LIN {X 0.147,Y -413.932,Z 942.824,A 0.000,B 0.000,C 90.000,E1 4.302} C_DIS
LIN {X -0.071,Y -420.578,Z 942.807,A 0.000,B 0.000,C 90.000,E1 1.260} C_DIS
LIN {X -0.166,Y -425.869,Z 942.795,A 0.000,B 0.000,C 90.000,E1 359.141} C_DIS
LIN {X 0.033,Y -428.792,Z 942.791,A 0.000,B 0.000,C 90.000,E1 358.282} C_DIS
LIN {X 0.078,Y -429.567,Z 942.790,A 0.000,B 0.000,C 90.000,E1 358.108} C_DIS
LIN {X -0.181,Y -431.033,Z 942.788,A 0.000,B 0.000,C 90.000,E1 357.879} C_DIS
LIN {X -0.110,Y -433.741,Z 942.786,A 0.000,B 0.000,C 90.000,E1 357.535} C_DIS
LIN {X -0.183,Y -435.827,Z 942.785,A 0.000,B 0.000,C 90.000,E1 357.306} C_DIS
LIN {X -0.171,Y -439.740,Z 942.783,A 0.000,B 0.000,C 90.000,E1 357.020} C_DIS
LIN {X -0.164,Y -441.464,Z 942.783,A 0.000,B 0.000,C 90.000,E1 356.906} C_DIS
LIN {X 0.019,Y -456.050,Z 942.779,A 0.000,B 0.000,C 90.000,E1 356.159} C_DIS
LIN {X -0.206,Y -464.593,Z 942.776,A 0.000,B 0.000,C 90.000,E1 355.755} C_DIS
LIN {X 0.207,Y -481.185,Z 942.771,A 0.000,B 0.000,C 90.000,E1 354.837} C_DIS
LIN {X 0.033,Y -494.438,Z 942.768,A 0.000,B 0.000,C 90.000,E1 354.147} C_DIS
LIN {X 0.171,Y -504.283,Z 942.764,A 0.000,B 0.000,C 90.000,E1 353.571} C_DIS
LIN {X -0.140,Y -515.374,Z 942.761,A 0.000,B 0.000,C 90.000,E1 352.932} C_DIS
LIN {X -0.046,Y -523.150,Z 942.758,A 0.000,B 0.000,C 90.000,E1 352.413} C_DIS
LIN {X -0.040,Y -531.958,Z 942.754,A 0.000,B 0.000,C 90.000,E1 351.781} C_DIS
LIN {X 0.025,Y -539.240,Z 942.751,A 0.000,B 0.000,C 90.000,E1 351.197} C_DIS
LIN {X -0.295,Y -546.239,Z 942.748,A 0.000,B 0.000,C 90.000,E1 350.622} C_DIS
LIN {X -0.106,Y -551.498,Z 942.745,A 0.000,B 0.000,C 90.000,E1 350.095} C_DIS
LIN {X 0.210,Y -557.779,Z 942.741,A 0.000,B 0.000,C 90.000,E1 349.398} C_DIS
LIN {X -0.265,Y -563.672,Z 942.737,A 0.000,B 0.000,C 90.000,E1 348.757} C_DIS
LIN {X 0.059,Y -568.140,Z 942.734,A 0.000,B 0.000,C 90.000,E1 348.173} C_DIS
LIN {X -0.068,Y -575.153,Z 942.729,A 0.000,B 0.000,C 90.000,E1 347.229} C_DIS
LIN {X 0.103,Y -579.773,Z 942.725,A 0.000,B 0.000,C 90.000,E1 346.533} C_DIS
LIN {X 0.025,Y -586.493,Z 942.719,A 0.000,B 0.000,C 90.000,E1 345.463} C_DIS
LIN {X 0.044,Y -592.545,Z 942.713,A 0.000,B 0.000,C 90.000,E1 344.393} C_DIS
LIN {X 0.209,Y -597.463,Z 942.708,A 0.000,B 0.000,C 90.000,E1 343.449} C_DIS
LIN {X 0.026,Y -601.982,Z 942.703,A 0.000,B 0.000,C 90.000,E1 342.543} C_DIS
LIN {X -0.139,Y -606.953,Z 942.697,A 0.000,B 0.000,C 90.000,E1 341.511} C_DIS
LIN {X -0.175,Y -610.557,Z 942.693,A 0.000,B 0.000,C 90.000,E1 340.732} C_DIS
LIN {X 0.025,Y -613.980,Z 942.689,A 0.000,B 0.000,C 90.000,E1 339.934} C_DIS
LIN {X 0.013,Y -618.273,Z 942.683,A 0.000,B 0.000,C 90.000,E1 338.901} C_DIS
LIN {X 0.283,Y -622.282,Z 942.677,A 0.000,B 0.000,C 90.000,E1 337.847} C_DIS
LIN {X 0.035,Y -626.049,Z 942.671,A 0.000,B 0.000,C 90.000,E1 336.847} C_DIS
LIN {X -0.400,Y -630.401,Z 942.664,A 0.000,B 0.000,C 90.000,E1 335.613} C_DIS
LIN {X 0.327,Y -634.450,Z 942.657,A 0.000,B 0.000,C 90.000,E1 334.280} C_DIS
LIN {X -0.012,Y -638.192,Z 942.650,A 0.000,B 0.000,C 90.000,E1 333.050} C_DIS
LIN {X 0.220,Y -640.863,Z 942.645,A 0.000,B 0.000,C 90.000,E1 332.025} C_DIS
LIN {X -0.152,Y -642.800,Z 942.641,A 0.000,B 0.000,C 90.000,E1 331.307} C_DIS
LIN {X 0.034,Y -646.291,Z 942.632,A 0.000,B 0.000,C 90.000,E1 329.793} C_DIS
LIN {X 0.199,Y -648.852,Z 942.625,A 0.000,B 0.000,C 90.000,E1 328.535} C_DIS
LIN {X 0.231,Y -650.232,Z 942.621,A 0.000,B 0.000,C 90.000,E1 327.788} C_DIS
LIN {X -0.186,Y -651.837,Z 942.616,A 0.000,B 0.000,C 90.000,E1 326.834} C_DIS
LIN {X -0.140,Y -653.569,Z 942.609,A 0.000,B 0.000,C 90.000,E1 325.595} C_DIS
LIN {X -0.149,Y -654.821,Z 942.603,A 0.000,B 0.000,C 90.000,E1 324.609} C_DIS
LIN {X -0.141,Y -655.872,Z 942.598,A 0.000,B 0.000,C 90.000,E1 323.623} C_DIS
LIN {X 0.286,Y -657.151,Z 942.590,A 0.000,B 0.000,C 90.000,E1 322.110} C_DIS
LIN {X -0.238,Y -658.485,Z 942.580,A 0.000,B 0.000,C 90.000,E1 320.436} C_DIS
LIN {X 0.159,Y -659.046,Z 942.576,A 0.000,B 0.000,C 90.000,E1 319.666} C_DIS
LIN {X 0.057,Y -660.436,Z 942.565,A 0.000,B 0.000,C 90.000,E1 317.715} C_DIS
LIN {X -0.058,Y -661.637,Z 942.557,A 0.000,B 0.000,C 90.000,E1 316.257} C_DIS
LIN {X 0.373,Y -662.239,Z 942.553,A 0.000,B 0.000,C 90.000,E1 315.486} C_DIS
LIN {X -0.195,Y -664.346,Z 942.539,A 0.000,B 0.000,C 90.000,E1 313.095} C_DIS
LIN {X -0.202,Y -665.986,Z 942.530,A 0.000,B 0.000,C 90.000,E1 311.391} C_DIS
LIN {X -0.170,Y -667.075,Z 942.523,A 0.000,B 0.000,C 90.000,E1 310.172} C_DIS
LIN {X -0.041,Y -668.319,Z 942.515,A 0.000,B 0.000,C 90.000,E1 308.705} C_DIS
LIN {X -0.404,Y -669.174,Z 942.508,A 0.000,B 0.000,C 90.000,E1 307.523} C_DIS
LIN {X 0.209,Y -669.600,Z 942.504,A 0.000,B 0.000,C 90.000,E1 306.744} C_DIS
LIN {X 0.390,Y -670.030,Z 942.498,A 0.000,B 0.000,C 90.000,E1 305.518} C_DIS
LIN {X 0.009,Y -670.808,Z 942.485,A 0.000,B 0.000,C 90.000,E1 303.372} C_DIS
LIN {X -0.049,Y -671.525,Z 942.477,A 0.000,B 0.000,C 90.000,E1 301.926} C_DIS
LIN {X -0.135,Y -675.368,Z 942.453,A 0.000,B 0.000,C 90.000,E1 297.590} C_DIS
LIN {X -0.137,Y -678.486,Z 942.443,A 0.000,B 0.000,C 90.000,E1 295.668} C_DIS
LIN {X -0.057,Y -680.495,Z 942.436,A 0.000,B 0.000,C 90.000,E1 294.463} C_DIS
LIN {X 0.046,Y -682.176,Z 942.429,A 0.000,B 0.000,C 90.000,E1 293.259} C_DIS
LIN {X 0.384,Y -682.822,Z 942.425,A 0.000,B 0.000,C 90.000,E1 292.514} C_DIS
LIN {X -0.104,Y -682.320,Z 942.423,A 0.000,B 0.000,C 90.000,E1 292.078} C_DIS
LIN {X -0.159,Y -681.925,Z 942.421,A 0.000,B 0.000,C 90.000,E1 291.844} C_DIS
LIN {X 0.038,Y -680.853,Z 942.420,A 0.000,B 0.000,C 90.000,E1 291.589} C_DIS
LIN {X 0.079,Y -678.846,Z 942.418,A 0.000,B 0.000,C 90.000,E1 291.227} C_DIS
LIN {X 0.172,Y -678.042,Z 942.417,A 0.000,B 0.000,C 90.000,E1 291.099} C_DIS
LIN {X 0.263,Y -676.847,Z 942.417,A 0.000,B 0.000,C 90.000,E1 290.972} C_DIS
LIN {X -0.270,Y -673.855,Z 942.415,A 0.000,B 0.000,C 90.000,E1 290.791} C_DIS
LIN {X -0.145,Y -669.235,Z 942.414,A 0.000,B 0.000,C 90.000,E1 290.482} C_DIS
LIN {X -0.196,Y -666.122,Z 942.413,A 0.000,B 0.000,C 90.000,E1 290.301} C_DIS
LIN {X 0.016,Y -663.674,Z 942.412,A 0.000,B 0.000,C 90.000,E1 290.120} C_DIS
LIN {X 0.198,Y -661.585,Z 942.411,A 0.000,B 0.000,C 90.000,E1 289.939} C_DIS
LIN {X 0.134,Y -661.564,Z 942.411,A 0.000,B 0.000,C 90.000,E1 289.939} C_DIS
LIN {X 0.203,Y -661.139,Z 942.410,A 0.000,B 0.000,C 90.000,E1 289.812} C_DIS
LIN {X 0.209,Y -661.461,Z 942.409,A 0.000,B 0.000,C 90.000,E1 289.523} C_DIS
LIN {X 0.322,Y -662.225,Z 942.407,A 0.000,B 0.000,C 90.000,E1 289.268} C_DIS
LIN {X 0.275,Y -663.656,Z 942.405,A 0.000,B 0.000,C 90.000,E1 288.906} C_DIS
LIN {X 0.104,Y -670.753,Z 942.398,A 0.000,B 0.000,C 90.000,E1 287.583} C_DIS
LIN {X 0.162,Y -673.111,Z 942.395,A 0.000,B 0.000,C 90.000,E1 287.094} C_DIS
LIN {X -0.022,Y -676.230,Z 942.391,A 0.000,B 0.000,C 90.000,E1 286.386} C_DIS
LIN {X 0.015,Y -678.639,Z 942.387,A 0.000,B 0.000,C 90.000,E1 285.662} C_DIS
LIN {X -0.071,Y -680.054,Z 942.384,A 0.000,B 0.000,C 90.000,E1 285.190} C_DIS
LIN {X -0.181,Y -681.680,Z 942.380,A 0.000,B 0.000,C 90.000,E1 284.481} C_DIS
LIN {X -0.301,Y -683.543,Z 942.375,A 0.000,B 0.000,C 90.000,E1 283.536} C_DIS
LIN {X 0.289,Y -684.620,Z 942.371,A 0.000,B 0.000,C 90.000,E1 282.771} C_DIS
LIN {X 0.197,Y -685.705,Z 942.366,A 0.000,B 0.000,C 90.000,E1 281.827} C_DIS
LIN {X -0.004,Y -685.932,Z 942.362,A 0.000,B 0.000,C 90.000,E1 281.130} C_DIS
LIN {X -0.048,Y -685.875,Z 942.359,A 0.000,B 0.000,C 90.000,E1 280.658} C_DIS
LIN {X -0.219,Y -685.455,Z 942.357,A 0.000,B 0.000,C 90.000,E1 280.197} C_DIS
LIN {X -0.271,Y -684.611,Z 942.354,A 0.000,B 0.000,C 90.000,E1 279.726} C_DIS
LIN {X 0.260,Y -684.093,Z 942.353,A 0.000,B 0.000,C 90.000,E1 279.443} C_DIS
LIN {X 0.195,Y -682.770,Z 942.350,A 0.000,B 0.000,C 90.000,E1 278.973} C_DIS
LIN {X 0.013,Y -681.051,Z 942.347,A 0.000,B 0.000,C 90.000,E1 278.511} C_DIS
LIN {X -0.177,Y -678.961,Z 942.345,A 0.000,B 0.000,C 90.000,E1 278.049} C_DIS
LIN {X 0.087,Y -673.637,Z 942.339,A 0.000,B 0.000,C 90.000,E1 276.947} C_DIS
LIN {X -0.232,Y -670.321,Z 942.335,A 0.000,B 0.000,C 90.000,E1 276.372} C_DIS
LIN {X 0.089,Y -666.532,Z 942.332,A 0.000,B 0.000,C 90.000,E1 275.739} C_DIS
LIN {X -0.194,Y -663.162,Z 942.329,A 0.000,B 0.000,C 90.000,E1 275.277} C_DIS
LIN {X 0.159,Y -659.351,Z 942.327,A 0.000,B 0.000,C 90.000,E1 274.759} C_DIS
LIN {X -0.319,Y -653.995,Z 942.323,A 0.000,B 0.000,C 90.000,E1 274.188} C_DIS
LIN {X -0.137,Y -648.110,Z 942.320,A 0.000,B 0.000,C 90.000,E1 273.555} C_DIS
LIN {X 0.241,Y -644.469,Z 942.318,A 0.000,B 0.000,C 90.000,E1 273.154} C_DIS
LIN {X 0.040,Y -637.861,Z 942.314,A 0.000,B 0.000,C 90.000,E1 272.579} C_DIS
LIN {X 0.156,Y -631.004,Z 942.311,A 0.000,B 0.000,C 90.000,E1 272.007} C_DIS
LIN {X 0.012,Y -623.443,Z 942.308,A 0.000,B 0.000,C 90.000,E1 271.489} C_DIS
LIN {X 0.226,Y -615.726,Z 942.306,A 0.000,B 0.000,C 90.000,E1 270.974} C_DIS
LIN {X 0.284,Y -611.147,Z 942.304,A 0.000,B 0.000,C 90.000,E1 270.688} C_DIS
LIN {X -0.126,Y -602.884,Z 942.302,A 0.000,B 0.000,C 90.000,E1 270.286} C_DIS
LIN {X 0.293,Y -597.983,Z 942.300,A 0.000,B 0.000,C 90.000,E1 270.000} C_DIS
LIN {X 0.177,Y -590.946,Z 942.299,A 0.000,B 0.000,C 90.000,E1 269.714} C_DIS
LIN {X -0.196,Y -583.749,Z 942.297,A 0.000,B 0.000,C 90.000,E1 269.484} C_DIS
LIN {X -0.179,Y -578.065,Z 942.296,A 0.000,B 0.000,C 90.000,E1 269.312} C_DIS
LIN {X 0.176,Y -569.943,Z 942.295,A 0.000,B 0.000,C 90.000,E1 269.083} C_DIS
LIN {X 0.222,Y -563.354,Z 942.294,A 0.000,B 0.000,C 90.000,E1 268.969} C_DIS
LIN {X 0.233,Y -559.044,Z 942.294,A 0.000,B 0.000,C 90.000,E1 268.912} C_DIS
LIN {X -0.170,Y -551.665,Z 942.294,A 0.000,B 0.000,C 90.000,E1 268.912} C_DIS
LIN {X -0.201,Y -548.189,Z 942.294,A 0.000,B 0.000,C 90.000,E1 268.854} C_DIS
LIN {X 0.006,Y -545.918,Z 942.293,A 0.000,B 0.000,C 90.000,E1 268.740} C_DIS
LIN {X -0.032,Y -545.812,Z 942.293,A 0.000,B 0.000,C 90.000,E1 268.740} C_DIS
LIN {X -0.003,Y -544.306,Z 942.292,A 0.000,B 0.000,C 90.000,E1 268.568} C_DIS
LIN {X -0.045,Y -544.268,Z 942.292,A 0.000,B 0.000,C 90.000,E1 268.568} C_DIS
LIN {X 0.209,Y -543.727,Z 942.290,A 0.000,B 0.000,C 90.000,E1 268.224} C_DIS
LIN {X -0.222,Y -542.695,Z 942.286,A 0.000,B 0.000,C 90.000,E1 267.421} C_DIS
LIN {X 0.132,Y -540.319,Z 942.270,A 0.000,B 0.000,C 90.000,E1 264.546} C_DIS
LIN {X 0.272,Y -539.546,Z 942.263,A 0.000,B 0.000,C 90.000,E1 263.394} C_DIS
LIN {X -0.088,Y -538.398,Z 942.254,A 0.000,B 0.000,C 90.000,E1 261.724} C_DIS
LIN {X 0.104,Y -537.716,Z 942.249,A 0.000,B 0.000,C 90.000,E1 260.849} C_DIS
LIN {X 0.204,Y -536.799,Z 942.245,A 0.000,B 0.000,C 90.000,E1 259.982} C_DIS
LIN {X -0.084,Y -535.189,Z 942.238,A 0.000,B 0.000,C 90.000,E1 258.870} C_DIS
LIN {X -0.241,Y -532.500,Z 942.227,A 0.000,B 0.000,C 90.000,E1 256.881} C_DIS
LIN {X 0.124,Y -530.513,Z 942.217,A 0.000,B 0.000,C 90.000,E1 255.117} C_DIS
LIN {X 0.208,Y -528.495,Z 942.208,A 0.000,B 0.000,C 90.000,E1 253.378} C_DIS
LIN {X 0.089,Y -526.789,Z 942.200,A 0.000,B 0.000,C 90.000,E1 251.945} C_DIS
LIN {X -0.235,Y -524.579,Z 942.190,A 0.000,B 0.000,C 90.000,E1 250.242} C_DIS
LIN {X 0.230,Y -521.965,Z 942.179,A 0.000,B 0.000,C 90.000,E1 248.156} C_DIS
LIN {X 0.014,Y -520.787,Z 942.174,A 0.000,B 0.000,C 90.000,E1 247.305} C_DIS
LIN {X 0.006,Y -518.625,Z 942.166,A 0.000,B 0.000,C 90.000,E1 245.845} C_DIS
LIN {X -0.248,Y -516.291,Z 942.158,A 0.000,B 0.000,C 90.000,E1 244.409} C_DIS
LIN {X 0.009,Y -514.428,Z 942.151,A 0.000,B 0.000,C 90.000,E1 243.204} C_DIS
LIN {X 0.118,Y -512.090,Z 942.143,A 0.000,B 0.000,C 90.000,E1 241.719} C_DIS
LIN {X -0.016,Y -509.635,Z 942.135,A 0.000,B 0.000,C 90.000,E1 240.255} C_DIS
LIN {X -0.078,Y -507.478,Z 942.128,A 0.000,B 0.000,C 90.000,E1 239.076} C_DIS
LIN {X 0.083,Y -505.103,Z 942.122,A 0.000,B 0.000,C 90.000,E1 237.867} C_DIS
LIN {X -0.217,Y -502.477,Z 942.115,A 0.000,B 0.000,C 90.000,E1 236.707} C_DIS
LIN {X 0.013,Y -499.011,Z 942.107,A 0.000,B 0.000,C 90.000,E1 235.182} C_DIS
LIN {X 0.034,Y -494.928,Z 942.097,A 0.000,B 0.000,C 90.000,E1 233.371} C_DIS
LIN {X 0.308,Y -491.653,Z 942.088,A 0.000,B 0.000,C 90.000,E1 231.823} C_DIS
LIN {X -0.161,Y -488.276,Z 942.080,A 0.000,B 0.000,C 90.000,E1 230.356} C_DIS
LIN {X 0.123,Y -484.079,Z 942.070,A 0.000,B 0.000,C 90.000,E1 228.485} C_DIS
LIN {X -0.170,Y -478.513,Z 942.056,A 0.000,B 0.000,C 90.000,E1 226.053} C_DIS
LIN {X -0.270,Y -475.011,Z 942.047,A 0.000,B 0.000,C 90.000,E1 224.514} C_DIS
LIN {X 0.134,Y -472.293,Z 942.040,A 0.000,B 0.000,C 90.000,E1 223.218} C_DIS
LIN {X 0.006,Y -468.191,Z 942.030,A 0.000,B 0.000,C 90.000,E1 221.353} C_DIS
LIN {X -0.013,Y -462.640,Z 942.016,A 0.000,B 0.000,C 90.000,E1 218.830} C_DIS
LIN {X 0.022,Y -459.198,Z 942.007,A 0.000,B 0.000,C 90.000,E1 217.237} C_DIS
LIN {X -0.016,Y -455.705,Z 941.998,A 0.000,B 0.000,C 90.000,E1 215.644} C_DIS
LIN {X 0.066,Y -451.487,Z 941.987,A 0.000,B 0.000,C 90.000,E1 213.706} C_DIS
LIN {X 0.108,Y -447.877,Z 941.978,A 0.000,B 0.000,C 90.000,E1 212.084} C_DIS
LIN {X 0.142,Y -443.620,Z 941.968,A 0.000,B 0.000,C 90.000,E1 210.129} C_DIS
LIN {X 0.186,Y -440.068,Z 941.958,A 0.000,B 0.000,C 90.000,E1 208.487} C_DIS
LIN {X -0.046,Y -436.559,Z 941.949,A 0.000,B 0.000,C 90.000,E1 206.873} C_DIS
LIN {X 0.041,Y -432.890,Z 941.940,A 0.000,B 0.000,C 90.000,E1 205.207} C_DIS
LIN {X 0.068,Y -428.497,Z 941.929,A 0.000,B 0.000,C 90.000,E1 203.206} C_DIS
LIN {X -0.168,Y -424.011,Z 941.918,A 0.000,B 0.000,C 90.000,E1 201.227} C_DIS
LIN {X -0.125,Y -419.636,Z 941.907,A 0.000,B 0.000,C 90.000,E1 199.195} C_DIS
LIN {X -0.075,Y -415.556,Z 941.895,A 0.000,B 0.000,C 90.000,E1 197.149} C_DIS
LIN {X 0.021,Y -412.134,Z 941.886,A 0.000,B 0.000,C 90.000,E1 195.426} C_DIS
LIN {X -0.071,Y -409.314,Z 941.878,A 0.000,B 0.000,C 90.000,E1 194.064} C_DIS
LIN {X -0.094,Y -403.790,Z 941.863,A 0.000,B 0.000,C 90.000,E1 191.299} C_DIS
LIN {X -0.108,Y -399.818,Z 941.851,A 0.000,B 0.000,C 90.000,E1 189.208} C_DIS
LIN {X 0.199,Y -396.450,Z 941.841,A 0.000,B 0.000,C 90.000,E1 187.409} C_DIS
LIN {X 0.152,Y -391.109,Z 941.826,A 0.000,B 0.000,C 90.000,E1 184.588} C_DIS
LIN {X 0.059,Y -385.167,Z 941.806,A 0.000,B 0.000,C 90.000,E1 181.031} C_DIS
LIN {X -0.147,Y -384.240,Z 941.802,A 0.000,B 0.000,C 90.000,E1 180.344} C_DIS
LIN {X 0.024,Y -383.524,Z 941.798,A 0.000,B 0.000,C 90.000,E1 179.599} C_DIS
LIN {X 0.130,Y -383.112,Z 941.793,A 0.000,B 0.000,C 90.000,E1 178.682} C_DIS
LIN {X -0.083,Y -383.293,Z 941.789,A 0.000,B 0.000,C 90.000,E1 177.993} C_DIS
LIN {X 0.018,Y -384.400,Z 941.784,A 0.000,B 0.000,C 90.000,E1 177.078} C_DIS
LIN {X -0.063,Y -385.223,Z 941.782,A 0.000,B 0.000,C 90.000,E1 176.731} C_DIS
LIN {X -0.043,Y -387.526,Z 941.779,A 0.000,B 0.000,C 90.000,E1 176.159} C_DIS
LIN {X -0.120,Y -389.435,Z 941.777,A 0.000,B 0.000,C 90.000,E1 175.812} C_DIS
LIN {X -0.085,Y -392.801,Z 941.774,A 0.000,B 0.000,C 90.000,E1 175.355} C_DIS
LIN {X 0.022,Y -397.374,Z 941.771,A 0.000,B 0.000,C 90.000,E1 174.837} C_DIS
LIN {X -0.101,Y -402.076,Z 941.769,A 0.000,B 0.000,C 90.000,E1 174.432} C_DIS
LIN {X 0.183,Y -414.801,Z 941.763,A 0.000,B 0.000,C 90.000,E1 173.337} C_DIS
LIN {X 0.071,Y -422.278,Z 941.760,A 0.000,B 0.000,C 90.000,E1 172.761} C_DIS
LIN {X 0.150,Y -433.139,Z 941.755,A 0.000,B 0.000,C 90.000,E1 171.837} C_DIS
LIN {X -0.096,Y -442.259,Z 941.750,A 0.000,B 0.000,C 90.000,E1 171.084} C_DIS
LIN {X 0.061,Y -449.669,Z 941.747,A 0.000,B 0.000,C 90.000,E1 170.387} C_DIS
LIN {X -0.251,Y -457.969,Z 941.742,A 0.000,B 0.000,C 90.000,E1 169.634} C_DIS
LIN {X -0.108,Y -466.514,Z 941.737,A 0.000,B 0.000,C 90.000,E1 168.757} C_DIS
LIN {X -0.110,Y -474.716,Z 941.733,A 0.000,B 0.000,C 90.000,E1 167.881} C_DIS
LIN {X -0.157,Y -479.909,Z 941.729,A 0.000,B 0.000,C 90.000,E1 167.285} C_DIS
LIN {X -0.114,Y -484.578,Z 941.726,A 0.000,B 0.000,C 90.000,E1 166.700} C_DIS
LIN {X -0.004,Y -489.361,Z 941.723,A 0.000,B 0.000,C 90.000,E1 166.117} C_DIS
LIN {X 0.294,Y -498.691,Z 941.716,A 0.000,B 0.000,C 90.000,E1 164.866} C_DIS
LIN {X -0.045,Y -508.142,Z 941.709,A 0.000,B 0.000,C 90.000,E1 163.559} C_DIS
LIN {X -0.059,Y -514.083,Z 941.704,A 0.000,B 0.000,C 90.000,E1 162.670} C_DIS
LIN {X -0.134,Y -517.012,Z 941.701,A 0.000,B 0.000,C 90.000,E1 162.236} C_DIS
LIN {X -0.230,Y -523.718,Z 941.696,A 0.000,B 0.000,C 90.000,E1 161.221} C_DIS
LIN {X -0.049,Y -532.822,Z 941.688,A 0.000,B 0.000,C 90.000,E1 159.752} C_DIS
LIN {X 0.012,Y -537.342,Z 941.684,A 0.000,B 0.000,C 90.000,E1 159.028} C_DIS
LIN {X -0.059,Y -545.963,Z 941.676,A 0.000,B 0.000,C 90.000,E1 157.614} C_DIS
LIN {X 0.079,Y -551.791,Z 941.670,A 0.000,B 0.000,C 90.000,E1 156.613} C_DIS
LIN {X 0.186,Y -558.101,Z 941.664,A 0.000,B 0.000,C 90.000,E1 155.485} C_DIS
LIN {X 0.171,Y -561.769,Z 941.660,A 0.000,B 0.000,C 90.000,E1 154.793} C_DIS
LIN {X -0.002,Y -566.757,Z 941.655,A 0.000,B 0.000,C 90.000,E1 153.845} C_DIS
LIN {X 0.136,Y -571.562,Z 941.649,A 0.000,B 0.000,C 90.000,E1 152.871} C_DIS
LIN {X 0.111,Y -577.600,Z 941.642,A 0.000,B 0.000,C 90.000,E1 151.513} C_DIS
LIN {X -0.194,Y -582.319,Z 941.636,A 0.000,B 0.000,C 90.000,E1 150.461} C_DIS
LIN {X 0.110,Y -588.834,Z 941.627,A 0.000,B 0.000,C 90.000,E1 148.820} C_DIS
LIN {X 0.174,Y -590.883,Z 941.624,A 0.000,B 0.000,C 90.000,E1 148.280} C_DIS
LIN {X 0.060,Y -595.772,Z 941.617,A 0.000,B 0.000,C 90.000,E1 146.962} C_DIS
LIN {X -0.194,Y -599.601,Z 941.611,A 0.000,B 0.000,C 90.000,E1 145.928} C_DIS
LIN {X 0.093,Y -603.366,Z 941.605,A 0.000,B 0.000,C 90.000,E1 144.848} C_DIS
LIN {X -0.208,Y -607.033,Z 941.599,A 0.000,B 0.000,C 90.000,E1 143.829} C_DIS
LIN {X -0.254,Y -612.461,Z 941.590,A 0.000,B 0.000,C 90.000,E1 142.271} C_DIS
LIN {X -0.301,Y -617.936,Z 941.582,A 0.000,B 0.000,C 90.000,E1 140.723} C_DIS
LIN {X -0.004,Y -621.603,Z 941.576,A 0.000,B 0.000,C 90.000,E1 139.666} C_DIS
LIN {X -0.066,Y -625.177,Z 941.570,A 0.000,B 0.000,C 90.000,E1 138.647} C_DIS
LIN {X -0.047,Y -631.997,Z 941.560,A 0.000,B 0.000,C 90.000,E1 136.863} C_DIS
LIN {X 0.309,Y -636.820,Z 941.553,A 0.000,B 0.000,C 90.000,E1 135.567} C_DIS
LIN {X -0.150,Y -641.548,Z 941.546,A 0.000,B 0.000,C 90.000,E1 134.352} C_DIS
LIN {X -0.208,Y -648.129,Z 941.537,A 0.000,B 0.000,C 90.000,E1 132.609} C_DIS
LIN {X 0.410,Y -653.792,Z 941.528,A 0.000,B 0.000,C 90.000,E1 131.067} C_DIS
LIN {X -0.170,Y -658.497,Z 941.522,A 0.000,B 0.000,C 90.000,E1 129.886} C_DIS
LIN {X 0.227,Y -664.114,Z 941.513,A 0.000,B 0.000,C 90.000,E1 128.382} C_DIS
LIN {X -0.115,Y -670.545,Z 941.504,A 0.000,B 0.000,C 90.000,E1 126.710} C_DIS
LIN {X 0.222,Y -675.653,Z 941.496,A 0.000,B 0.000,C 90.000,E1 125.231} C_DIS
LIN {X 0.123,Y -678.822,Z 941.491,A 0.000,B 0.000,C 90.000,E1 124.278} C_DIS
LIN {X -0.108,Y -681.051,Z 941.487,A 0.000,B 0.000,C 90.000,E1 123.579} C_DIS
LIN {X -0.133,Y -683.774,Z 941.481,A 0.000,B 0.000,C 90.000,E1 122.625} C_DIS
LIN {X 0.253,Y -685.677,Z 941.477,A 0.000,B 0.000,C 90.000,E1 121.878} C_DIS
LIN {X -0.090,Y -688.397,Z 941.471,A 0.000,B 0.000,C 90.000,E1 120.718} C_DIS
LIN {X -0.241,Y -689.369,Z 941.468,A 0.000,B 0.000,C 90.000,E1 120.256} C_DIS
LIN {X -0.154,Y -690.686,Z 941.464,A 0.000,B 0.000,C 90.000,E1 119.539} C_DIS
LIN {X -0.051,Y -691.866,Z 941.460,A 0.000,B 0.000,C 90.000,E1 118.821} C_DIS
LIN {X 0.308,Y -693.091,Z 941.455,A 0.000,B 0.000,C 90.000,E1 117.847} C_DIS
LIN {X 0.064,Y -693.963,Z 941.450,A 0.000,B 0.000,C 90.000,E1 116.924} C_DIS
LIN {X 0.131,Y -694.382,Z 941.444,A 0.000,B 0.000,C 90.000,E1 115.976} C_DIS
LIN {X 0.210,Y -694.574,Z 941.439,A 0.000,B 0.000,C 90.000,E1 115.027} C_DIS
LIN {X 0.041,Y -694.545,Z 941.435,A 0.000,B 0.000,C 90.000,E1 114.335} C_DIS
LIN {X -0.377,Y -694.333,Z 941.433,A 0.000,B 0.000,C 90.000,E1 113.898} C_DIS
LIN {X 0.118,Y -693.575,Z 941.430,A 0.000,B 0.000,C 90.000,E1 113.387} C_DIS
LIN {X 0.089,Y -692.962,Z 941.429,A 0.000,B 0.000,C 90.000,E1 113.153} C_DIS
LIN {X -0.305,Y -691.978,Z 941.427,A 0.000,B 0.000,C 90.000,E1 112.950} C_DIS
LIN {X -0.214,Y -690.152,Z 941.425,A 0.000,B 0.000,C 90.000,E1 112.589} C_DIS
LIN {X -0.097,Y -689.148,Z 941.425,A 0.000,B 0.000,C 90.000,E1 112.461} C_DIS
LIN {X 0.153,Y -684.795,Z 941.423,A 0.000,B 0.000,C 90.000,E1 112.099} C_DIS
LIN {X 0.180,Y -681.659,Z 941.422,A 0.000,B 0.000,C 90.000,E1 111.897} C_DIS
LIN {X -0.220,Y -677.447,Z 941.421,A 0.000,B 0.000,C 90.000,E1 111.770} C_DIS
LIN {X -0.163,Y -672.043,Z 941.420,A 0.000,B 0.000,C 90.000,E1 111.663} C_DIS
LIN {X -0.195,Y -667.270,Z 941.420,A 0.000,B 0.000,C 90.000,E1 111.589} C_DIS
LIN {X 0.222,Y -661.340,Z 941.420,A 0.000,B 0.000,C 90.000,E1 111.535} C_DIS
LIN {X 0.150,Y -636.856,Z 941.420,A 0.000,B 0.000,C 90.000,E1 111.535} C_DIS
LIN {X -0.260,Y -632.899,Z 941.420,A 0.000,B 0.000,C 90.000,E1 111.535} C_DIS
LIN {X 0.229,Y -627.205,Z 941.419,A 0.000,B 0.000,C 90.000,E1 111.408} C_DIS
LIN {X 0.341,Y -621.437,Z 941.418,A 0.000,B 0.000,C 90.000,E1 111.280} C_DIS
LIN {X 0.134,Y -614.374,Z 941.417,A 0.000,B 0.000,C 90.000,E1 111.099} C_DIS
LIN {X 0.072,Y -608.017,Z 941.416,A 0.000,B 0.000,C 90.000,E1 110.865} C_DIS
LIN {X 0.218,Y -601.707,Z 941.414,A 0.000,B 0.000,C 90.000,E1 110.556} C_DIS
LIN {X 0.248,Y -595.200,Z 941.412,A 0.000,B 0.000,C 90.000,E1 110.174} C_DIS
LIN {X -0.215,Y -578.416,Z 941.406,A 0.000,B 0.000,C 90.000,E1 109.033} C_DIS
LIN {X -0.024,Y -576.781,Z 941.405,A 0.000,B 0.000,C 90.000,E1 108.906} C_DIS
LIN {X 0.235,Y -568.253,Z 941.403,A 0.000,B 0.000,C 90.000,E1 108.417} C_DIS
LIN {X 0.157,Y -562.882,Z 941.401,A 0.000,B 0.000,C 90.000,E1 108.181} C_DIS
LIN {X 0.270,Y -555.097,Z 941.399,A 0.000,B 0.000,C 90.000,E1 107.819} C_DIS
LIN {X 0.027,Y -553.556,Z 941.399,A 0.000,B 0.000,C 90.000,E1 107.764} C_DIS
LIN {X -0.091,Y -552.007,Z 941.398,A 0.000,B 0.000,C 90.000,E1 107.638} C_DIS
LIN {X -0.121,Y -551.987,Z 941.398,A 0.000,B 0.000,C 90.000,E1 107.638} C_DIS
LIN {X 0.172,Y -551.611,Z 941.396,A 0.000,B 0.000,C 90.000,E1 107.330} C_DIS
LIN {X 0.031,Y -552.325,Z 941.385,A 0.000,B 0.000,C 90.000,E1 105.245} C_DIS
LIN {X 0.034,Y -553.405,Z 941.372,A 0.000,B 0.000,C 90.000,E1 103.008} C_DIS
LIN {X -0.296,Y -554.554,Z 941.363,A 0.000,B 0.000,C 90.000,E1 101.366} C_DIS
LIN {X -0.067,Y -555.932,Z 941.354,A 0.000,B 0.000,C 90.000,E1 99.670} C_DIS
LIN {X -0.049,Y -557.138,Z 941.346,A 0.000,B 0.000,C 90.000,E1 98.276} C_DIS
LIN {X -0.091,Y -558.228,Z 941.338,A 0.000,B 0.000,C 90.000,E1 96.891} C_DIS
LIN {X -0.169,Y -559.198,Z 941.331,A 0.000,B 0.000,C 90.000,E1 95.511} C_DIS
LIN {X -0.223,Y -560.000,Z 941.323,A 0.000,B 0.000,C 90.000,E1 94.131} C_DIS
LIN {X -0.271,Y -560.799,Z 941.315,A 0.000,B 0.000,C 90.000,E1 92.751} C_DIS
LIN {X -0.244,Y -561.526,Z 941.306,A 0.000,B 0.000,C 90.000,E1 91.088} C_DIS
LIN {X 0.251,Y -562.064,Z 941.298,A 0.000,B 0.000,C 90.000,E1 89.656} C_DIS
LIN {X -0.255,Y -562.441,Z 941.289,A 0.000,B 0.000,C 90.000,E1 88.051} C_DIS
LIN {X 0.143,Y -562.720,Z 941.283,A 0.000,B 0.000,C 90.000,E1 86.906} C_DIS
LIN {X 0.233,Y -563.000,Z 941.274,A 0.000,B 0.000,C 90.000,E1 85.241} C_DIS
LIN {X -0.182,Y -563.219,Z 941.265,A 0.000,B 0.000,C 90.000,E1 83.628} C_DIS
LIN {X -0.283,Y -563.652,Z 941.252,A 0.000,B 0.000,C 90.000,E1 81.432} C_DIS
LIN {X -0.189,Y -564.454,Z 941.240,A 0.000,B 0.000,C 90.000,E1 79.218} C_DIS
LIN {X -0.191,Y -565.001,Z 941.234,A 0.000,B 0.000,C 90.000,E1 78.117} C_DIS
LIN {X 0.217,Y -565.735,Z 941.226,A 0.000,B 0.000,C 90.000,E1 76.700} C_DIS
LIN {X 0.099,Y -566.615,Z 941.219,A 0.000,B 0.000,C 90.000,E1 75.338} C_DIS
LIN {X 0.163,Y -567.608,Z 941.209,A 0.000,B 0.000,C 90.000,E1 73.685} C_DIS
LIN {X 0.020,Y -568.560,Z 941.200,A 0.000,B 0.000,C 90.000,E1 72.054} C_DIS
LIN {X -0.096,Y -569.406,Z 941.191,A 0.000,B 0.000,C 90.000,E1 70.423} C_DIS
LIN {X -0.173,Y -569.802,Z 941.185,A 0.000,B 0.000,C 90.000,E1 69.337} C_DIS
LIN {X -0.227,Y -570.262,Z 941.178,A 0.000,B 0.000,C 90.000,E1 67.975} C_DIS
LIN {X -0.096,Y -570.663,Z 941.167,A 0.000,B 0.000,C 90.000,E1 66.049} C_DIS
LIN {X 0.092,Y -570.946,Z 941.159,A 0.000,B 0.000,C 90.000,E1 64.665} C_DIS
LIN {X 0.019,Y -571.159,Z 941.152,A 0.000,B 0.000,C 90.000,E1 63.307} C_DIS
LIN {X 0.299,Y -571.238,Z 941.143,A 0.000,B 0.000,C 90.000,E1 61.641} C_DIS
LIN {X -0.156,Y -571.245,Z 941.134,A 0.000,B 0.000,C 90.000,E1 60.049} C_DIS
LIN {X -0.062,Y -571.362,Z 941.128,A 0.000,B 0.000,C 90.000,E1 58.948} C_DIS
LIN {X -0.170,Y -571.239,Z 941.121,A 0.000,B 0.000,C 90.000,E1 57.867} C_DIS
LIN {X -0.153,Y -570.927,Z 941.114,A 0.000,B 0.000,C 90.000,E1 56.501} C_DIS
LIN {X 0.179,Y -570.369,Z 941.106,A 0.000,B 0.000,C 90.000,E1 55.102} C_DIS
LIN {X -0.090,Y -569.842,Z 941.100,A 0.000,B 0.000,C 90.000,E1 54.036} C_DIS
LIN {X 0.090,Y -569.126,Z 941.094,A 0.000,B 0.000,C 90.000,E1 52.924} C_DIS
LIN {X 0.144,Y -568.074,Z 941.088,A 0.000,B 0.000,C 90.000,E1 51.823} C_DIS
LIN {X 0.068,Y -567.225,Z 941.083,A 0.000,B 0.000,C 90.000,E1 51.009} C_DIS
LIN {X -0.016,Y -566.236,Z 941.079,A 0.000,B 0.000,C 90.000,E1 50.194} C_DIS
LIN {X -0.007,Y -564.611,Z 941.073,A 0.000,B 0.000,C 90.000,E1 49.094} C_DIS
LIN {X 0.146,Y -563.747,Z 941.070,A 0.000,B 0.000,C 90.000,E1 48.528} C_DIS
LIN {X -0.310,Y -561.571,Z 941.064,A 0.000,B 0.000,C 90.000,E1 47.472} C_DIS
LIN {X -0.170,Y -560.422,Z 941.061,A 0.000,B 0.000,C 90.000,E1 46.905} C_DIS
LIN {X 0.038,Y -558.378,Z 941.056,A 0.000,B 0.000,C 90.000,E1 46.053} C_DIS
LIN {X -0.179,Y -556.127,Z 941.051,A 0.000,B 0.000,C 90.000,E1 45.243} C_DIS
LIN {X -0.073,Y -554.483,Z 941.048,A 0.000,B 0.000,C 90.000,E1 44.676} C_DIS
LIN {X -0.330,Y -551.699,Z 941.044,A 0.000,B 0.000,C 90.000,E1 43.866} C_DIS
LIN {X -0.217,Y -548.587,Z 941.039,A 0.000,B 0.000,C 90.000,E1 43.014} C_DIS
LIN {X 0.196,Y -547.547,Z 941.037,A 0.000,B 0.000,C 90.000,E1 42.690} C_DIS
LIN {X 0.064,Y -544.568,Z 941.033,A 0.000,B 0.000,C 90.000,E1 42.000} C_DIS
LIN {X -0.094,Y -541.308,Z 941.029,A 0.000,B 0.000,C 90.000,E1 41.310} C_DIS
LIN {X -0.097,Y -535.446,Z 941.023,A 0.000,B 0.000,C 90.000,E1 40.172} C_DIS
LIN {X 0.070,Y -531.302,Z 941.019,A 0.000,B 0.000,C 90.000,E1 39.439} C_DIS
LIN {X -0.235,Y -525.270,Z 941.014,A 0.000,B 0.000,C 90.000,E1 38.463} C_DIS
LIN {X -0.163,Y -520.639,Z 941.010,A 0.000,B 0.000,C 90.000,E1 37.729} C_DIS
LIN {X -0.263,Y -516.779,Z 941.006,A 0.000,B 0.000,C 90.000,E1 37.156} C_DIS
LIN {X -0.049,Y -510.658,Z 941.001,A 0.000,B 0.000,C 90.000,E1 36.251} C_DIS
LIN {X 0.078,Y -506.347,Z 940.998,A 0.000,B 0.000,C 90.000,E1 35.644} C_DIS
LIN {X 0.283,Y -501.804,Z 940.995,A 0.000,B 0.000,C 90.000,E1 35.025} C_DIS
LIN {X -0.098,Y -495.537,Z 940.991,A 0.000,B 0.000,C 90.000,E1 34.326} C_DIS
LIN {X 0.235,Y -493.001,Z 940.989,A 0.000,B 0.000,C 90.000,E1 33.992} C_DIS
LIN {X -0.105,Y -486.092,Z 940.985,A 0.000,B 0.000,C 90.000,E1 33.293} C_DIS
LIN {X -0.131,Y -483.377,Z 940.983,A 0.000,B 0.000,C 90.000,E1 33.007} C_DIS
LIN {X 0.219,Y -474.758,Z 940.979,A 0.000,B 0.000,C 90.000,E1 32.133} C_DIS
LIN {X 0.075,Y -466.009,Z 940.974,A 0.000,B 0.000,C 90.000,E1 31.337} C_DIS
LIN {X 0.084,Y -460.034,Z 940.971,A 0.000,B 0.000,C 90.000,E1 30.797} C_DIS
LIN {X 0.131,Y -449.349,Z 940.966,A 0.000,B 0.000,C 90.000,E1 29.873} C_DIS
LIN {X 0.064,Y -443.148,Z 940.963,A 0.000,B 0.000,C 90.000,E1 29.361} C_DIS
LIN {X -0.108,Y -428.050,Z 940.956,A 0.000,B 0.000,C 90.000,E1 28.103} C_DIS
LIN {X -0.052,Y -405.905,Z 940.945,A 0.000,B 0.000,C 90.000,E1 26.027} C_DIS
LIN {X -0.111,Y -398.655,Z 940.940,A 0.000,B 0.000,C 90.000,E1 25.283} C_DIS
LIN {X 0.054,Y -396.164,Z 940.939,A 0.000,B 0.000,C 90.000,E1 24.975} C_DIS
LIN {X -0.027,Y -394.967,Z 940.938,A 0.000,B 0.000,C 90.000,E1 24.823} C_DIS
LIN {X -0.226,Y -391.800,Z 940.935,A 0.000,B 0.000,C 90.000,E1 24.335} C_DIS
LIN {X 0.012,Y -390.405,Z 940.933,A 0.000,B 0.000,C 90.000,E1 23.898} C_DIS
LIN {X -0.080,Y -390.061,Z 940.932,A 0.000,B 0.000,C 90.000,E1 23.823} C_DIS
LIN {X -0.121,Y -389.219,Z 940.929,A 0.000,B 0.000,C 90.000,E1 23.206} C_DIS
LIN {X -0.018,Y -389.211,Z 940.924,A 0.000,B 0.000,C 90.000,E1 22.280} C_DIS
LIN {X -0.132,Y -389.839,Z 940.918,A 0.000,B 0.000,C 90.000,E1 21.227} C_DIS
LIN {X 0.032,Y -392.926,Z 940.900,A 0.000,B 0.000,C 90.000,E1 18.000} C_DIS
LIN {X -0.071,Y -395.816,Z 940.886,A 0.000,B 0.000,C 90.000,E1 15.536} C_DIS
LIN {X 0.040,Y -399.584,Z 940.871,A 0.000,B 0.000,C 90.000,E1 12.703} C_DIS
LIN {X 0.030,Y -404.448,Z 940.853,A 0.000,B 0.000,C 90.000,E1 9.557} C_DIS
LIN {X 0.023,Y -408.048,Z 940.842,A 0.000,B 0.000,C 90.000,E1 7.473} C_DIS
LIN {X 0.137,Y -414.656,Z 940.822,A 0.000,B 0.000,C 90.000,E1 4.012} C_DIS
LIN {X -0.047,Y -422.206,Z 940.804,A 0.000,B 0.000,C 90.000,E1 0.630} C_DIS
LIN {X 0.209,Y -425.023,Z 940.797,A 0.000,B 0.000,C 90.000,E1 359.427} C_DIS
LIN {X -0.166,Y -425.935,Z 940.795,A 0.000,B 0.000,C 90.000,E1 359.141} C_DIS
LIN {X -0.056,Y -428.112,Z 940.791,A 0.000,B 0.000,C 90.000,E1 358.453} C_DIS
LIN {X 0.053,Y -430.295,Z 940.789,A 0.000,B 0.000,C 90.000,E1 357.936} C_DIS
LIN {X 0.088,Y -431.194,Z 940.788,A 0.000,B 0.000,C 90.000,E1 357.764} C_DIS
LIN {X 0.197,Y -433.737,Z 940.786,A 0.000,B 0.000,C 90.000,E1 357.421} C_DIS
LIN {X 0.071,Y -435.890,Z 940.784,A 0.000,B 0.000,C 90.000,E1 357.192} C_DIS
LIN {X 0.029,Y -440.730,Z 940.783,A 0.000,B 0.000,C 90.000,E1 356.846} C_DIS
LIN {X -0.055,Y -448.784,Z 940.780,A 0.000,B 0.000,C 90.000,E1 356.445} C_DIS
LIN {X 0.120,Y -458.928,Z 940.778,A 0.000,B 0.000,C 90.000,E1 355.927} C_DIS
LIN {X 0.126,Y -465.652,Z 940.776,A 0.000,B 0.000,C 90.000,E1 355.584} C_DIS
LIN {X 0.056,Y -482.280,Z 940.771,A 0.000,B 0.000,C 90.000,E1 354.723} C_DIS
LIN {X -0.026,Y -492.238,Z 940.768,A 0.000,B 0.000,C 90.000,E1 354.204} C_DIS
LIN {X 0.056,Y -505.244,Z 940.764,A 0.000,B 0.000,C 90.000,E1 353.457} C_DIS
LIN {X 0.067,Y -514.792,Z 940.760,A 0.000,B 0.000,C 90.000,E1 352.875} C_DIS
LIN {X 0.154,Y -522.665,Z 940.758,A 0.000,B 0.000,C 90.000,E1 352.356} C_DIS
LIN {X -0.047,Y -531.757,Z 940.754,A 0.000,B 0.000,C 90.000,E1 351.724} C_DIS
LIN {X 0.058,Y -539.031,Z 940.751,A 0.000,B 0.000,C 90.000,E1 351.141} C_DIS
LIN {X -0.168,Y -546.057,Z 940.747,A 0.000,B 0.000,C 90.000,E1 350.557} C_DIS
LIN {X -0.060,Y -551.379,Z 940.745,A 0.000,B 0.000,C 90.000,E1 350.038} C_DIS
LIN {X -0.123,Y -556.540,Z 940.742,A 0.000,B 0.000,C 90.000,E1 349.511} C_DIS
LIN {X -0.067,Y -562.496,Z 940.738,A 0.000,B 0.000,C 90.000,E1 348.814} C_DIS
LIN {X 0.001,Y -568.111,Z 940.734,A 0.000,B 0.000,C 90.000,E1 348.117} C_DIS
LIN {X -0.201,Y -572.179,Z 940.731,A 0.000,B 0.000,C 90.000,E1 347.589} C_DIS
LIN {X 0.072,Y -577.038,Z 940.727,A 0.000,B 0.000,C 90.000,E1 346.881} C_DIS
LIN {X -0.169,Y -581.517,Z 940.723,A 0.000,B 0.000,C 90.000,E1 346.228} C_DIS
LIN {X -0.131,Y -587.337,Z 940.718,A 0.000,B 0.000,C 90.000,E1 345.283} C_DIS
LIN {X -0.025,Y -592.613,Z 940.713,A 0.000,B 0.000,C 90.000,E1 344.338} C_DIS
LIN {X 0.307,Y -597.576,Z 940.708,A 0.000,B 0.000,C 90.000,E1 343.378} C_DIS
LIN {X -0.099,Y -602.705,Z 940.702,A 0.000,B 0.000,C 90.000,E1 342.362} C_DIS
LIN {X 0.321,Y -607.706,Z 940.696,A 0.000,B 0.000,C 90.000,E1 341.275} C_DIS
LIN {X 0.233,Y -612.458,Z 940.690,A 0.000,B 0.000,C 90.000,E1 340.242} C_DIS
LIN {X 0.202,Y -616.884,Z 940.685,A 0.000,B 0.000,C 90.000,E1 339.209} C_DIS
LIN {X -0.125,Y -620.993,Z 940.679,A 0.000,B 0.000,C 90.000,E1 338.209} C_DIS
LIN {X 0.189,Y -623.953,Z 940.675,A 0.000,B 0.000,C 90.000,E1 337.411} C_DIS
LIN {X -0.276,Y -628.453,Z 940.668,A 0.000,B 0.000,C 90.000,E1 336.177} C_DIS
LIN {X -0.187,Y -631.845,Z 940.662,A 0.000,B 0.000,C 90.000,E1 335.153} C_DIS
LIN {X -0.316,Y -635.111,Z 940.656,A 0.000,B 0.000,C 90.000,E1 334.152} C_DIS
LIN {X -0.078,Y -638.791,Z 940.649,A 0.000,B 0.000,C 90.000,E1 332.871} C_DIS
LIN {X -0.283,Y -642.793,Z 940.641,A 0.000,B 0.000,C 90.000,E1 331.385} C_DIS
LIN {X -0.029,Y -646.879,Z 940.631,A 0.000,B 0.000,C 90.000,E1 329.616} C_DIS
LIN {X -0.078,Y -649.396,Z 940.624,A 0.000,B 0.000,C 90.000,E1 328.377} C_DIS
LIN {X -0.384,Y -650.773,Z 940.620,A 0.000,B 0.000,C 90.000,E1 327.661} C_DIS
LIN {X 0.105,Y -652.343,Z 940.615,A 0.000,B 0.000,C 90.000,E1 326.628} C_DIS
LIN {X 0.160,Y -654.053,Z 940.608,A 0.000,B 0.000,C 90.000,E1 325.388} C_DIS
LIN {X -0.298,Y -655.572,Z 940.601,A 0.000,B 0.000,C 90.000,E1 324.196} C_DIS
LIN {X -0.285,Y -656.549,Z 940.596,A 0.000,B 0.000,C 90.000,E1 323.210} C_DIS
LIN {X -0.320,Y -657.584,Z 940.589,A 0.000,B 0.000,C 90.000,E1 321.984} C_DIS
LIN {X 0.046,Y -659.113,Z 940.578,A 0.000,B 0.000,C 90.000,E1 319.989} C_DIS
LIN {X -0.064,Y -660.169,Z 940.570,A 0.000,B 0.000,C 90.000,E1 318.528} C_DIS
LIN {X -0.148,Y -661.362,Z 940.561,A 0.000,B 0.000,C 90.000,E1 317.067} C_DIS
LIN {X 0.239,Y -662.554,Z 940.553,A 0.000,B 0.000,C 90.000,E1 315.567} C_DIS
LIN {X -0.328,Y -664.880,Z 940.538,A 0.000,B 0.000,C 90.000,E1 312.933} C_DIS
LIN {X 0.122,Y -666.290,Z 940.530,A 0.000,B 0.000,C 90.000,E1 311.434} C_DIS
LIN {X -0.282,Y -667.384,Z 940.524,A 0.000,B 0.000,C 90.000,E1 310.253} C_DIS
LIN {X 0.274,Y -668.656,Z 940.515,A 0.000,B 0.000,C 90.000,E1 308.749} C_DIS
LIN {X -0.090,Y -669.543,Z 940.509,A 0.000,B 0.000,C 90.000,E1 307.569} C_DIS
LIN {X -0.416,Y -669.987,Z 940.505,A 0.000,B 0.000,C 90.000,E1 306.870} C_DIS
LIN {X 0.310,Y -670.425,Z 940.498,A 0.000,B 0.000,C 90.000,E1 305.598} C_DIS
LIN {X -0.200,Y -671.085,Z 940.487,A 0.000,B 0.000,C 90.000,E1 303.706} C_DIS
LIN {X -0.100,Y -671.910,Z 940.478,A 0.000,B 0.000,C 90.000,E1 302.005} C_DIS
LIN {X 0.353,Y -676.049,Z 940.452,A 0.000,B 0.000,C 90.000,E1 297.385} C_DIS
LIN {X 0.361,Y -679.175,Z 940.442,A 0.000,B 0.000,C 90.000,E1 295.463} C_DIS
LIN {X 0.166,Y -681.126,Z 940.435,A 0.000,B 0.000,C 90.000,E1 294.283} C_DIS
LIN {X 0.079,Y -682.452,Z 940.430,A 0.000,B 0.000,C 90.000,E1 293.334} C_DIS
LIN {X -0.205,Y -683.116,Z 940.426,A 0.000,B 0.000,C 90.000,E1 292.642} C_DIS
LIN {X -0.003,Y -682.988,Z 940.424,A 0.000,B 0.000,C 90.000,E1 292.386} C_DIS
LIN {X 0.143,Y -682.411,Z 940.422,A 0.000,B 0.000,C 90.000,E1 291.897} C_DIS
LIN {X 0.090,Y -681.524,Z 940.420,A 0.000,B 0.000,C 90.000,E1 291.663} C_DIS
LIN {X -0.403,Y -678.783,Z 940.418,A 0.000,B 0.000,C 90.000,E1 291.227} C_DIS
LIN {X -0.310,Y -677.866,Z 940.417,A 0.000,B 0.000,C 90.000,E1 291.099} C_DIS
LIN {X -0.217,Y -676.519,Z 940.416,A 0.000,B 0.000,C 90.000,E1 290.972} C_DIS
LIN {X -0.217,Y -670.209,Z 940.414,A 0.000,B 0.000,C 90.000,E1 290.556} C_DIS
LIN {X -0.088,Y -664.116,Z 940.412,A 0.000,B 0.000,C 90.000,E1 290.174} C_DIS
LIN {X -0.070,Y -661.940,Z 940.411,A 0.000,B 0.000,C 90.000,E1 289.993} C_DIS
LIN {X -0.109,Y -661.921,Z 940.411,A 0.000,B 0.000,C 90.000,E1 289.993} C_DIS
LIN {X 0.190,Y -661.417,Z 940.410,A 0.000,B 0.000,C 90.000,E1 289.812} C_DIS
LIN {X 0.317,Y -661.915,Z 940.408,A 0.000,B 0.000,C 90.000,E1 289.450} C_DIS
LIN {X 0.325,Y -663.698,Z 940.406,A 0.000,B 0.000,C 90.000,E1 288.960} C_DIS
LIN {X 0.152,Y -670.770,Z 940.398,A 0.000,B 0.000,C 90.000,E1 287.638} C_DIS
LIN {X 0.142,Y -674.213,Z 940.394,A 0.000,B 0.000,C 90.000,E1 286.913} C_DIS
LIN {X 0.022,Y -676.309,Z 940.391,A 0.000,B 0.000,C 90.000,E1 286.441} C_DIS
LIN {X 0.057,Y -678.738,Z 940.387,A 0.000,B 0.000,C 90.000,E1 285.717} C_DIS
LIN {X -0.030,Y -680.159,Z 940.385,A 0.000,B 0.000,C 90.000,E1 285.245} C_DIS
LIN {X -0.141,Y -681.823,Z 940.381,A 0.000,B 0.000,C 90.000,E1 284.537} C_DIS
LIN {X -0.262,Y -683.699,Z 940.375,A 0.000,B 0.000,C 90.000,E1 283.592} C_DIS
LIN {X 0.329,Y -684.823,Z 940.371,A 0.000,B 0.000,C 90.000,E1 282.827} C_DIS
LIN {X 0.096,Y -685.924,Z 940.366,A 0.000,B 0.000,C 90.000,E1 281.895} C_DIS
LIN {X 0.036,Y -686.243,Z 940.362,A 0.000,B 0.000,C 90.000,E1 281.186} C_DIS
LIN {X -0.007,Y -686.210,Z 940.360,A 0.000,B 0.000,C 90.000,E1 280.715} C_DIS
LIN {X -0.178,Y -685.812,Z 940.357,A 0.000,B 0.000,C 90.000,E1 280.254} C_DIS
LIN {X -0.203,Y -685.490,Z 940.356,A 0.000,B 0.000,C 90.000,E1 280.018} C_DIS
LIN {X 0.304,Y -684.569,Z 940.353,A 0.000,B 0.000,C 90.000,E1 279.500} C_DIS
LIN {X 0.241,Y -683.246,Z 940.350,A 0.000,B 0.000,C 90.000,E1 279.029} C_DIS
LIN {X 0.060,Y -681.556,Z 940.348,A 0.000,B 0.000,C 90.000,E1 278.568} C_DIS
LIN {X -0.127,Y -679.501,Z 940.345,A 0.000,B 0.000,C 90.000,E1 278.106} C_DIS
LIN {X 0.287,Y -676.007,Z 940.341,A 0.000,B 0.000,C 90.000,E1 277.352} C_DIS
LIN {X -0.011,Y -672.914,Z 940.338,A 0.000,B 0.000,C 90.000,E1 276.777} C_DIS
LIN {X -0.252,Y -670.220,Z 940.335,A 0.000,B 0.000,C 90.000,E1 276.315} C_DIS
LIN {X 0.070,Y -666.405,Z 940.332,A 0.000,B 0.000,C 90.000,E1 275.682} C_DIS
LIN {X -0.125,Y -663.939,Z 940.330,A 0.000,B 0.000,C 90.000,E1 275.334} C_DIS
LIN {X 0.139,Y -659.157,Z 940.326,A 0.000,B 0.000,C 90.000,E1 274.702} C_DIS
LIN {X -0.242,Y -654.943,Z 940.323,A 0.000,B 0.000,C 90.000,E1 274.245} C_DIS
LIN {X -0.053,Y -649.118,Z 940.320,A 0.000,B 0.000,C 90.000,E1 273.612} C_DIS
LIN {X 0.282,Y -644.231,Z 940.317,A 0.000,B 0.000,C 90.000,E1 273.094} C_DIS
LIN {X 0.122,Y -637.647,Z 940.314,A 0.000,B 0.000,C 90.000,E1 272.522} C_DIS
LIN {X 0.224,Y -630.704,Z 940.311,A 0.000,B 0.000,C 90.000,E1 271.949} C_DIS
LIN {X 0.195,Y -623.239,Z 940.308,A 0.000,B 0.000,C 90.000,E1 271.432} C_DIS
LIN {X 0.252,Y -617.145,Z 940.306,A 0.000,B 0.000,C 90.000,E1 271.031} C_DIS
LIN {X -0.148,Y -610.879,Z 940.304,A 0.000,B 0.000,C 90.000,E1 270.688} C_DIS
LIN {X 0.013,Y -602.497,Z 940.301,A 0.000,B 0.000,C 90.000,E1 270.229} C_DIS
LIN {X -0.195,Y -597.459,Z 940.300,A 0.000,B 0.000,C 90.000,E1 270.000} C_DIS
LIN {X 0.258,Y -590.259,Z 940.298,A 0.000,B 0.000,C 90.000,E1 269.656} C_DIS
LIN {X -0.040,Y -584.954,Z 940.297,A 0.000,B 0.000,C 90.000,E1 269.484} C_DIS
LIN {X -0.017,Y -577.348,Z 940.296,A 0.000,B 0.000,C 90.000,E1 269.255} C_DIS
LIN {X -0.275,Y -571.633,Z 940.295,A 0.000,B 0.000,C 90.000,E1 269.141} C_DIS
LIN {X 0.233,Y -564.977,Z 940.294,A 0.000,B 0.000,C 90.000,E1 268.969} C_DIS
LIN {X -0.042,Y -558.598,Z 940.294,A 0.000,B 0.000,C 90.000,E1 268.912} C_DIS
LIN {X 0.269,Y -553.935,Z 940.294,A 0.000,B 0.000,C 90.000,E1 268.854} C_DIS
LIN {X 0.024,Y -550.952,Z 940.294,A 0.000,B 0.000,C 90.000,E1 268.854} C_DIS
LIN {X 0.053,Y -547.897,Z 940.293,A 0.000,B 0.000,C 90.000,E1 268.797} C_DIS
LIN {X 0.015,Y -547.866,Z 940.293,A 0.000,B 0.000,C 90.000,E1 268.797} C_DIS
LIN {X 0.254,Y -544.089,Z 940.291,A 0.000,B 0.000,C 90.000,E1 268.339} C_DIS
LIN {X 0.213,Y -544.070,Z 940.291,A 0.000,B 0.000,C 90.000,E1 268.339} C_DIS
LIN {X -0.124,Y -543.049,Z 940.287,A 0.000,B 0.000,C 90.000,E1 267.650} C_DIS
LIN {X 0.261,Y -540.354,Z 940.270,A 0.000,B 0.000,C 90.000,E1 264.489} C_DIS
LIN {X -0.136,Y -539.578,Z 940.263,A 0.000,B 0.000,C 90.000,E1 263.394} C_DIS
LIN {X 0.116,Y -538.452,Z 940.254,A 0.000,B 0.000,C 90.000,E1 261.659} C_DIS
LIN {X 0.229,Y -537.768,Z 940.249,A 0.000,B 0.000,C 90.000,E1 260.792} C_DIS
LIN {X -0.201,Y -536.863,Z 940.244,A 0.000,B 0.000,C 90.000,E1 259.982} C_DIS
LIN {X 0.039,Y -535.215,Z 940.238,A 0.000,B 0.000,C 90.000,E1 258.814} C_DIS
LIN {X -0.122,Y -532.511,Z 940.227,A 0.000,B 0.000,C 90.000,E1 256.825} C_DIS
LIN {X -0.137,Y -530.517,Z 940.217,A 0.000,B 0.000,C 90.000,E1 255.102} C_DIS
LIN {X -0.188,Y -528.476,Z 940.208,A 0.000,B 0.000,C 90.000,E1 253.378} C_DIS
LIN {X -0.307,Y -526.767,Z 940.200,A 0.000,B 0.000,C 90.000,E1 251.945} C_DIS
LIN {X -0.136,Y -524.573,Z 940.190,A 0.000,B 0.000,C 90.000,E1 250.188} C_DIS
LIN {X 0.164,Y -522.325,Z 940.180,A 0.000,B 0.000,C 90.000,E1 248.411} C_DIS
LIN {X 0.150,Y -521.196,Z 940.175,A 0.000,B 0.000,C 90.000,E1 247.539} C_DIS
LIN {X 0.089,Y -518.593,Z 940.166,A 0.000,B 0.000,C 90.000,E1 245.793} C_DIS
LIN {X 0.180,Y -515.803,Z 940.156,A 0.000,B 0.000,C 90.000,E1 244.024} C_DIS
LIN {X -0.025,Y -513.000,Z 940.146,A 0.000,B 0.000,C 90.000,E1 242.281} C_DIS
LIN {X -0.032,Y -511.091,Z 940.139,A 0.000,B 0.000,C 90.000,E1 241.101} C_DIS
LIN {X 0.011,Y -508.508,Z 940.131,A 0.000,B 0.000,C 90.000,E1 239.616} C_DIS
LIN {X 0.187,Y -506.250,Z 940.125,A 0.000,B 0.000,C 90.000,E1 238.408} C_DIS
LIN {X -0.099,Y -503.759,Z 940.118,A 0.000,B 0.000,C 90.000,E1 237.248} C_DIS
LIN {X -0.245,Y -499.644,Z 940.108,A 0.000,B 0.000,C 90.000,E1 235.468} C_DIS
LIN {X 0.084,Y -495.538,Z 940.098,A 0.000,B 0.000,C 90.000,E1 233.623} C_DIS
LIN {X -0.073,Y -491.599,Z 940.088,A 0.000,B 0.000,C 90.000,E1 231.823} C_DIS
LIN {X 0.148,Y -488.229,Z 940.079,A 0.000,B 0.000,C 90.000,E1 230.275} C_DIS
LIN {X -0.116,Y -483.322,Z 940.068,A 0.000,B 0.000,C 90.000,E1 228.162} C_DIS
LIN {X 0.134,Y -478.461,Z 940.056,A 0.000,B 0.000,C 90.000,E1 225.972} C_DIS
LIN {X 0.239,Y -473.656,Z 940.043,A 0.000,B 0.000,C 90.000,E1 223.785} C_DIS
LIN {X 0.223,Y -468.838,Z 940.031,A 0.000,B 0.000,C 90.000,E1 221.595} C_DIS
LIN {X 0.115,Y -463.941,Z 940.019,A 0.000,B 0.000,C 90.000,E1 219.402} C_DIS
LIN {X 0.169,Y -460.534,Z 940.010,A 0.000,B 0.000,C 90.000,E1 217.810} C_DIS
LIN {X 0.158,Y -457.063,Z 940.001,A 0.000,B 0.000,C 90.000,E1 216.217} C_DIS
LIN {X 0.178,Y -453.585,Z 939.992,A 0.000,B 0.000,C 90.000,E1 214.612} C_DIS
LIN {X 0.083,Y -451.441,Z 939.987,A 0.000,B 0.000,C 90.000,E1 213.658} C_DIS
LIN {X -0.010,Y -447.853,Z 939.978,A 0.000,B 0.000,C 90.000,E1 212.054} C_DIS
LIN {X -0.210,Y -443.600,Z 939.967,A 0.000,B 0.000,C 90.000,E1 210.129} C_DIS
LIN {X -0.122,Y -439.342,Z 939.956,A 0.000,B 0.000,C 90.000,E1 208.153} C_DIS
LIN {X -0.004,Y -436.540,Z 939.949,A 0.000,B 0.000,C 90.000,E1 206.821} C_DIS
LIN {X 0.089,Y -432.115,Z 939.938,A 0.000,B 0.000,C 90.000,E1 204.823} C_DIS
LIN {X -0.083,Y -429.219,Z 939.931,A 0.000,B 0.000,C 90.000,E1 203.515} C_DIS
LIN {X -0.102,Y -425.490,Z 939.921,A 0.000,B 0.000,C 90.000,E1 201.844} C_DIS
LIN {X -0.017,Y -421.073,Z 939.910,A 0.000,B 0.000,C 90.000,E1 199.812} C_DIS
LIN {X -0.009,Y -415.576,Z 939.895,A 0.000,B 0.000,C 90.000,E1 197.094} C_DIS
LIN {X 0.089,Y -412.157,Z 939.885,A 0.000,B 0.000,C 90.000,E1 195.371} C_DIS
LIN {X 0.118,Y -408.575,Z 939.876,A 0.000,B 0.000,C 90.000,E1 193.647} C_DIS
LIN {X -0.020,Y -403.796,Z 939.862,A 0.000,B 0.000,C 90.000,E1 191.243} C_DIS
LIN {X -0.032,Y -399.825,Z 939.851,A 0.000,B 0.000,C 90.000,E1 189.151} C_DIS
LIN {X -0.118,Y -396.441,Z 939.841,A 0.000,B 0.000,C 90.000,E1 187.409} C_DIS
LIN {X -0.161,Y -391.055,Z 939.825,A 0.000,B 0.000,C 90.000,E1 184.588} C_DIS
LIN {X 0.031,Y -384.512,Z 939.804,A 0.000,B 0.000,C 90.000,E1 180.630} C_DIS
LIN {X 0.095,Y -383.271,Z 939.798,A 0.000,B 0.000,C 90.000,E1 179.542} C_DIS
LIN {X -0.127,Y -382.743,Z 939.794,A 0.000,B 0.000,C 90.000,E1 178.854} C_DIS
LIN {X -0.018,Y -382.763,Z 939.789,A 0.000,B 0.000,C 90.000,E1 177.936} C_DIS
LIN {X -0.190,Y -383.229,Z 939.786,A 0.000,B 0.000,C 90.000,E1 177.421} C_DIS
LIN {X 0.077,Y -383.464,Z 939.784,A 0.000,B 0.000,C 90.000,E1 177.020} C_DIS
LIN {X -0.041,Y -384.523,Z 939.781,A 0.000,B 0.000,C 90.000,E1 176.502} C_DIS
LIN {X -0.086,Y -386.045,Z 939.778,A 0.000,B 0.000,C 90.000,E1 176.102} C_DIS
LIN {X -0.170,Y -387.633,Z 939.776,A 0.000,B 0.000,C 90.000,E1 175.755} C_DIS
LIN {X -0.055,Y -389.118,Z 939.775,A 0.000,B 0.000,C 90.000,E1 175.469} C_DIS
LIN {X 0.036,Y -393.037,Z 939.772,A 0.000,B 0.000,C 90.000,E1 174.951} C_DIS
LIN {X -0.176,Y -395.845,Z 939.770,A 0.000,B 0.000,C 90.000,E1 174.666} C_DIS
LIN {X 0.050,Y -400.480,Z 939.768,A 0.000,B 0.000,C 90.000,E1 174.204} C_DIS
LIN {X -0.015,Y -419.802,Z 939.759,A 0.000,B 0.000,C 90.000,E1 172.648} C_DIS
LIN {X 0.033,Y -427.486,Z 939.756,A 0.000,B 0.000,C 90.000,E1 172.008} C_DIS
LIN {X 0.098,Y -438.394,Z 939.751,A 0.000,B 0.000,C 90.000,E1 171.084} C_DIS
LIN {X 0.069,Y -444.338,Z 939.748,A 0.000,B 0.000,C 90.000,E1 170.566} C_DIS
LIN {X 0.049,Y -453.256,Z 939.743,A 0.000,B 0.000,C 90.000,E1 169.746} C_DIS
LIN {X 0.069,Y -460.360,Z 939.739,A 0.000,B 0.000,C 90.000,E1 169.050} C_DIS
LIN {X 0.218,Y -466.104,Z 939.736,A 0.000,B 0.000,C 90.000,E1 168.465} C_DIS
LIN {X 0.064,Y -472.974,Z 939.732,A 0.000,B 0.000,C 90.000,E1 167.757} C_DIS
LIN {X 0.114,Y -479.441,Z 939.728,A 0.000,B 0.000,C 90.000,E1 166.992} C_DIS
LIN {X -0.077,Y -489.539,Z 939.721,A 0.000,B 0.000,C 90.000,E1 165.811} C_DIS
LIN {X -0.161,Y -497.697,Z 939.715,A 0.000,B 0.000,C 90.000,E1 164.755} C_DIS
LIN {X -0.221,Y -506.245,Z 939.709,A 0.000,B 0.000,C 90.000,E1 163.559} C_DIS
LIN {X -0.154,Y -514.306,Z 939.702,A 0.000,B 0.000,C 90.000,E1 162.362} C_DIS
LIN {X -0.195,Y -518.976,Z 939.698,A 0.000,B 0.000,C 90.000,E1 161.638} C_DIS
LIN {X 0.152,Y -521.944,Z 939.695,A 0.000,B 0.000,C 90.000,E1 161.167} C_DIS
LIN {X 0.147,Y -531.963,Z 939.687,A 0.000,B 0.000,C 90.000,E1 159.571} C_DIS
LIN {X 0.200,Y -536.587,Z 939.683,A 0.000,B 0.000,C 90.000,E1 158.847} C_DIS
LIN {X 0.084,Y -543.482,Z 939.676,A 0.000,B 0.000,C 90.000,E1 157.720} C_DIS
LIN {X -0.262,Y -550.987,Z 939.669,A 0.000,B 0.000,C 90.000,E1 156.485} C_DIS
LIN {X -0.060,Y -556.607,Z 939.664,A 0.000,B 0.000,C 90.000,E1 155.485} C_DIS
LIN {X -0.089,Y -560.349,Z 939.660,A 0.000,B 0.000,C 90.000,E1 154.793} C_DIS
LIN {X -0.033,Y -565.426,Z 939.655,A 0.000,B 0.000,C 90.000,E1 153.819} C_DIS
LIN {X -0.250,Y -570.863,Z 939.648,A 0.000,B 0.000,C 90.000,E1 152.743} C_DIS
LIN {X -0.135,Y -575.807,Z 939.642,A 0.000,B 0.000,C 90.000,E1 151.641} C_DIS
LIN {X 0.044,Y -580.636,Z 939.636,A 0.000,B 0.000,C 90.000,E1 150.539} C_DIS
LIN {X -0.190,Y -587.273,Z 939.627,A 0.000,B 0.000,C 90.000,E1 148.948} C_DIS
LIN {X 0.050,Y -590.340,Z 939.623,A 0.000,B 0.000,C 90.000,E1 148.122} C_DIS
LIN {X 0.108,Y -595.321,Z 939.616,A 0.000,B 0.000,C 90.000,E1 146.786} C_DIS
LIN {X -0.054,Y -598.319,Z 939.611,A 0.000,B 0.000,C 90.000,E1 146.008} C_DIS
LIN {X 0.122,Y -604.956,Z 939.601,A 0.000,B 0.000,C 90.000,E1 144.149} C_DIS
LIN {X -0.181,Y -611.268,Z 939.591,A 0.000,B 0.000,C 90.000,E1 142.351} C_DIS
LIN {X -0.255,Y -616.827,Z 939.582,A 0.000,B 0.000,C 90.000,E1 140.803} C_DIS
LIN {X 0.340,Y -621.424,Z 939.575,A 0.000,B 0.000,C 90.000,E1 139.461} C_DIS
LIN {X 0.066,Y -629.976,Z 939.562,A 0.000,B 0.000,C 90.000,E1 137.187} C_DIS
LIN {X 0.384,Y -634.907,Z 939.555,A 0.000,B 0.000,C 90.000,E1 135.891} C_DIS
LIN {X -0.195,Y -640.626,Z 939.547,A 0.000,B 0.000,C 90.000,E1 134.433} C_DIS
LIN {X -0.273,Y -647.263,Z 939.537,A 0.000,B 0.000,C 90.000,E1 132.690} C_DIS
LIN {X 0.329,Y -652.956,Z 939.529,A 0.000,B 0.000,C 90.000,E1 131.148} C_DIS
LIN {X 0.157,Y -657.665,Z 939.522,A 0.000,B 0.000,C 90.000,E1 129.930} C_DIS
LIN {X 0.117,Y -663.289,Z 939.514,A 0.000,B 0.000,C 90.000,E1 128.463} C_DIS
LIN {X -0.295,Y -666.966,Z 939.508,A 0.000,B 0.000,C 90.000,E1 127.523} C_DIS
LIN {X 0.274,Y -670.559,Z 939.503,A 0.000,B 0.000,C 90.000,E1 126.503} C_DIS
LIN {X 0.085,Y -674.929,Z 939.496,A 0.000,B 0.000,C 90.000,E1 125.311} C_DIS
LIN {X -0.037,Y -678.880,Z 939.490,A 0.000,B 0.000,C 90.000,E1 124.119} C_DIS
LIN {X 0.295,Y -681.128,Z 939.486,A 0.000,B 0.000,C 90.000,E1 123.372} C_DIS
LIN {X -0.109,Y -684.416,Z 939.479,A 0.000,B 0.000,C 90.000,E1 122.212} C_DIS
LIN {X 0.075,Y -685.615,Z 939.476,A 0.000,B 0.000,C 90.000,E1 121.720} C_DIS
LIN {X 0.117,Y -687.250,Z 939.472,A 0.000,B 0.000,C 90.000,E1 121.003} C_DIS
LIN {X -0.409,Y -688.789,Z 939.468,A 0.000,B 0.000,C 90.000,E1 120.335} C_DIS
LIN {X 0.245,Y -690.513,Z 939.463,A 0.000,B 0.000,C 90.000,E1 119.333} C_DIS
LIN {X 0.344,Y -691.665,Z 939.459,A 0.000,B 0.000,C 90.000,E1 118.615} C_DIS
LIN {X -0.237,Y -692.811,Z 939.454,A 0.000,B 0.000,C 90.000,E1 117.719} C_DIS
LIN {X 0.133,Y -693.597,Z 939.449,A 0.000,B 0.000,C 90.000,E1 116.744} C_DIS
LIN {X 0.201,Y -693.968,Z 939.443,A 0.000,B 0.000,C 90.000,E1 115.796} C_DIS
LIN {X -0.351,Y -694.056,Z 939.438,A 0.000,B 0.000,C 90.000,E1 114.899} C_DIS
LIN {X -0.277,Y -693.916,Z 939.433,A 0.000,B 0.000,C 90.000,E1 113.951} C_DIS
LIN {X -0.063,Y -693.220,Z 939.430,A 0.000,B 0.000,C 90.000,E1 113.462} C_DIS
LIN {X 0.180,Y -692.713,Z 939.429,A 0.000,B 0.000,C 90.000,E1 113.206} C_DIS
LIN {X -0.246,Y -690.747,Z 939.426,A 0.000,B 0.000,C 90.000,E1 112.770} C_DIS
LIN {X -0.128,Y -690.148,Z 939.426,A 0.000,B 0.000,C 90.000,E1 112.642} C_DIS
LIN {X -0.012,Y -689.297,Z 939.425,A 0.000,B 0.000,C 90.000,E1 112.514} C_DIS
LIN {X 0.102,Y -688.026,Z 939.424,A 0.000,B 0.000,C 90.000,E1 112.386} C_DIS
LIN {X -0.099,Y -682.376,Z 939.422,A 0.000,B 0.000,C 90.000,E1 111.972} C_DIS
LIN {X 0.169,Y -680.195,Z 939.422,A 0.000,B 0.000,C 90.000,E1 111.844} C_DIS
LIN {X 0.138,Y -678.120,Z 939.421,A 0.000,B 0.000,C 90.000,E1 111.770} C_DIS
LIN {X -0.145,Y -675.522,Z 939.421,A 0.000,B 0.000,C 90.000,E1 111.716} C_DIS
LIN {X -0.231,Y -667.923,Z 939.420,A 0.000,B 0.000,C 90.000,E1 111.589} C_DIS
LIN {X 0.018,Y -660.371,Z 939.420,A 0.000,B 0.000,C 90.000,E1 111.535} C_DIS
LIN {X -0.046,Y -637.394,Z 939.420,A 0.000,B 0.000,C 90.000,E1 111.535} C_DIS
LIN {X -0.234,Y -634.886,Z 939.420,A 0.000,B 0.000,C 90.000,E1 111.535} C_DIS
LIN {X -0.131,Y -626.740,Z 939.419,A 0.000,B 0.000,C 90.000,E1 111.408} C_DIS
LIN {X -0.067,Y -620.982,Z 939.418,A 0.000,B 0.000,C 90.000,E1 111.280} C_DIS
LIN {X 0.225,Y -615.436,Z 939.417,A 0.000,B 0.000,C 90.000,E1 111.099} C_DIS
LIN {X -0.019,Y -608.488,Z 939.416,A 0.000,B 0.000,C 90.000,E1 110.865} C_DIS
LIN {X -0.161,Y -601.210,Z 939.414,A 0.000,B 0.000,C 90.000,E1 110.536} C_DIS
LIN {X -0.152,Y -596.170,Z 939.412,A 0.000,B 0.000,C 90.000,E1 110.248} C_DIS
LIN {X 0.257,Y -585.153,Z 939.408,A 0.000,B 0.000,C 90.000,E1 109.450} C_DIS
LIN {X 0.069,Y -578.102,Z 939.405,A 0.000,B 0.000,C 90.000,E1 108.960} C_DIS
LIN {X 0.045,Y -569.680,Z 939.403,A 0.000,B 0.000,C 90.000,E1 108.489} C_DIS
LIN {X 0.070,Y -565.992,Z 939.402,A 0.000,B 0.000,C 90.000,E1 108.308} C_DIS
LIN {X -0.078,Y -555.730,Z 939.399,A 0.000,B 0.000,C 90.000,E1 107.873} C_DIS
LIN {X -0.237,Y -554.252,Z 939.399,A 0.000,B 0.000,C 90.000,E1 107.819} C_DIS
LIN {X 0.150,Y -552.466,Z 939.398,A 0.000,B 0.000,C 90.000,E1 107.638} C_DIS
LIN {X -0.235,Y -552.045,Z 939.398,A 0.000,B 0.000,C 90.000,E1 107.638} C_DIS
LIN {X 0.237,Y -552.020,Z 939.398,A 0.000,B 0.000,C 90.000,E1 107.583} C_DIS
LIN {X 0.138,Y -551.796,Z 939.397,A 0.000,B 0.000,C 90.000,E1 107.457} C_DIS
LIN {X -0.022,Y -551.799,Z 939.394,A 0.000,B 0.000,C 90.000,E1 106.913} C_DIS
LIN {X -0.130,Y -552.460,Z 939.385,A 0.000,B 0.000,C 90.000,E1 105.245} C_DIS
LIN {X 0.172,Y -553.237,Z 939.375,A 0.000,B 0.000,C 90.000,E1 103.536} C_DIS
LIN {X 0.076,Y -554.510,Z 939.365,A 0.000,B 0.000,C 90.000,E1 101.591} C_DIS
LIN {X -0.219,Y -556.063,Z 939.354,A 0.000,B 0.000,C 90.000,E1 99.670} C_DIS
LIN {X -0.145,Y -557.465,Z 939.344,A 0.000,B 0.000,C 90.000,E1 97.992} C_DIS
LIN {X -0.173,Y -558.517,Z 939.337,A 0.000,B 0.000,C 90.000,E1 96.606} C_DIS
LIN {X 0.240,Y -559.280,Z 939.331,A 0.000,B 0.000,C 90.000,E1 95.454} C_DIS
LIN {X 0.189,Y -560.073,Z 939.323,A 0.000,B 0.000,C 90.000,E1 94.073} C_DIS
LIN {X 0.145,Y -560.874,Z 939.315,A 0.000,B 0.000,C 90.000,E1 92.694} C_DIS
LIN {X 0.271,Y -561.723,Z 939.304,A 0.000,B 0.000,C 90.000,E1 90.745} C_DIS
LIN {X 0.208,Y -562.210,Z 939.297,A 0.000,B 0.000,C 90.000,E1 89.370} C_DIS
LIN {X 0.266,Y -562.551,Z 939.287,A 0.000,B 0.000,C 90.000,E1 87.707} C_DIS
LIN {X 0.132,Y -562.803,Z 939.281,A 0.000,B 0.000,C 90.000,E1 86.617} C_DIS
LIN {X 0.092,Y -563.056,Z 939.274,A 0.000,B 0.000,C 90.000,E1 85.241} C_DIS
LIN {X 0.150,Y -563.225,Z 939.266,A 0.000,B 0.000,C 90.000,E1 83.856} C_DIS
LIN {X 0.223,Y -563.444,Z 939.258,A 0.000,B 0.000,C 90.000,E1 82.470} C_DIS
LIN {X 0.062,Y -563.964,Z 939.248,A 0.000,B 0.000,C 90.000,E1 80.557} C_DIS
LIN {X 0.230,Y -564.520,Z 939.240,A 0.000,B 0.000,C 90.000,E1 79.162} C_DIS
LIN {X -0.042,Y -565.178,Z 939.232,A 0.000,B 0.000,C 90.000,E1 77.813} C_DIS
LIN {X 0.082,Y -565.803,Z 939.226,A 0.000,B 0.000,C 90.000,E1 76.700} C_DIS
LIN {X 0.135,Y -566.845,Z 939.217,A 0.000,B 0.000,C 90.000,E1 75.046} C_DIS
LIN {X -0.188,Y -567.818,Z 939.208,A 0.000,B 0.000,C 90.000,E1 73.433} C_DIS
LIN {X 0.049,Y -568.734,Z 939.199,A 0.000,B 0.000,C 90.000,E1 71.764} C_DIS
LIN {X -0.228,Y -569.421,Z 939.191,A 0.000,B 0.000,C 90.000,E1 70.423} C_DIS
LIN {X -0.103,Y -569.809,Z 939.185,A 0.000,B 0.000,C 90.000,E1 69.316} C_DIS
LIN {X 0.170,Y -570.241,Z 939.177,A 0.000,B 0.000,C 90.000,E1 67.922} C_DIS
LIN {X -0.227,Y -570.645,Z 939.167,A 0.000,B 0.000,C 90.000,E1 66.049} C_DIS
LIN {X -0.041,Y -570.915,Z 939.159,A 0.000,B 0.000,C 90.000,E1 64.665} C_DIS
LIN {X -0.113,Y -571.134,Z 939.152,A 0.000,B 0.000,C 90.000,E1 63.307} C_DIS
LIN {X 0.165,Y -571.201,Z 939.143,A 0.000,B 0.000,C 90.000,E1 61.641} C_DIS
LIN {X 0.034,Y -571.217,Z 939.132,A 0.000,B 0.000,C 90.000,E1 59.744} C_DIS
LIN {X -0.197,Y -571.284,Z 939.127,A 0.000,B 0.000,C 90.000,E1 58.948} C_DIS
LIN {X -0.306,Y -571.149,Z 939.121,A 0.000,B 0.000,C 90.000,E1 57.867} C_DIS
LIN {X -0.290,Y -570.813,Z 939.114,A 0.000,B 0.000,C 90.000,E1 56.501} C_DIS
LIN {X -0.221,Y -570.479,Z 939.109,A 0.000,B 0.000,C 90.000,E1 55.674} C_DIS
LIN {X -0.029,Y -569.991,Z 939.103,A 0.000,B 0.000,C 90.000,E1 54.562} C_DIS
LIN {X -0.180,Y -569.162,Z 939.096,A 0.000,B 0.000,C 90.000,E1 53.210} C_DIS
LIN {X -0.002,Y -567.845,Z 939.088,A 0.000,B 0.000,C 90.000,E1 51.823} C_DIS
LIN {X -0.080,Y -566.978,Z 939.083,A 0.000,B 0.000,C 90.000,E1 51.009} C_DIS
LIN {X -0.054,Y -565.555,Z 939.077,A 0.000,B 0.000,C 90.000,E1 49.908} C_DIS
LIN {X -0.160,Y -564.317,Z 939.073,A 0.000,B 0.000,C 90.000,E1 49.094} C_DIS
LIN {X -0.009,Y -563.425,Z 939.070,A 0.000,B 0.000,C 90.000,E1 48.528} C_DIS
LIN {X -0.003,Y -560.636,Z 939.062,A 0.000,B 0.000,C 90.000,E1 47.148} C_DIS
LIN {X 0.206,Y -558.669,Z 939.057,A 0.000,B 0.000,C 90.000,E1 46.296} C_DIS
LIN {X -0.010,Y -556.469,Z 939.053,A 0.000,B 0.000,C 90.000,E1 45.486} C_DIS
LIN {X -0.246,Y -553.978,Z 939.048,A 0.000,B 0.000,C 90.000,E1 44.676} C_DIS
LIN {X -0.156,Y -552.155,Z 939.045,A 0.000,B 0.000,C 90.000,E1 44.109} C_DIS
LIN {X -0.039,Y -549.094,Z 939.040,A 0.000,B 0.000,C 90.000,E1 43.257} C_DIS
LIN {X 0.013,Y -546.919,Z 939.037,A 0.000,B 0.000,C 90.000,E1 42.690} C_DIS
LIN {X -0.123,Y -543.903,Z 939.033,A 0.000,B 0.000,C 90.000,E1 42.000} C_DIS
LIN {X -0.286,Y -540.548,Z 939.029,A 0.000,B 0.000,C 90.000,E1 41.310} C_DIS
LIN {X -0.127,Y -535.392,Z 939.024,A 0.000,B 0.000,C 90.000,E1 40.297} C_DIS
LIN {X 0.038,Y -531.304,Z 939.020,A 0.000,B 0.000,C 90.000,E1 39.564} C_DIS
LIN {X 0.286,Y -524.319,Z 939.013,A 0.000,B 0.000,C 90.000,E1 38.382} C_DIS
LIN {X 0.026,Y -519.628,Z 939.009,A 0.000,B 0.000,C 90.000,E1 37.684} C_DIS
LIN {X 0.233,Y -515.706,Z 939.006,A 0.000,B 0.000,C 90.000,E1 37.076} C_DIS
LIN {X 0.095,Y -511.576,Z 939.003,A 0.000,B 0.000,C 90.000,E1 36.503} C_DIS
LIN {X -0.071,Y -507.322,Z 939.000,A 0.000,B 0.000,C 90.000,E1 35.931} C_DIS
LIN {X -0.055,Y -501.674,Z 938.995,A 0.000,B 0.000,C 90.000,E1 35.185} C_DIS
LIN {X 0.200,Y -495.338,Z 938.991,A 0.000,B 0.000,C 90.000,E1 34.405} C_DIS
LIN {X -0.136,Y -491.337,Z 938.989,A 0.000,B 0.000,C 90.000,E1 33.992} C_DIS
LIN {X -0.028,Y -486.062,Z 938.986,A 0.000,B 0.000,C 90.000,E1 33.420} C_DIS
LIN {X 0.105,Y -480.446,Z 938.983,A 0.000,B 0.000,C 90.000,E1 32.832} C_DIS
LIN {X 0.192,Y -471.933,Z 938.978,A 0.000,B 0.000,C 90.000,E1 32.005} C_DIS
LIN {X -0.040,Y -461.505,Z 938.973,A 0.000,B 0.000,C 90.000,E1 31.082} C_DIS
LIN {X 0.255,Y -450.834,Z 938.968,A 0.000,B 0.000,C 90.000,E1 30.129} C_DIS
LIN {X -0.134,Y -443.238,Z 938.964,A 0.000,B 0.000,C 90.000,E1 29.539} C_DIS
LIN {X -0.049,Y -427.962,Z 938.957,A 0.000,B 0.000,C 90.000,E1 28.231} C_DIS
LIN {X -0.042,Y -405.696,Z 938.945,A 0.000,B 0.000,C 90.000,E1 26.155} C_DIS
LIN {X 0.226,Y -397.023,Z 938.940,A 0.000,B 0.000,C 90.000,E1 25.207} C_DIS
LIN {X 0.104,Y -394.502,Z 938.938,A 0.000,B 0.000,C 90.000,E1 24.899} C_DIS
LIN {X -0.018,Y -391.434,Z 938.936,A 0.000,B 0.000,C 90.000,E1 24.387} C_DIS
LIN {X 0.195,Y -389.751,Z 938.933,A 0.000,B 0.000,C 90.000,E1 23.823} C_DIS
LIN {X -0.170,Y -389.117,Z 938.930,A 0.000,B 0.000,C 90.000,E1 23.334} C_DIS
LIN {X -0.094,Y -389.168,Z 938.924,A 0.000,B 0.000,C 90.000,E1 22.386} C_DIS
LIN {X 0.149,Y -389.808,Z 938.918,A 0.000,B 0.000,C 90.000,E1 21.280} C_DIS
LIN {X -0.066,Y -392.935,Z 938.901,A 0.000,B 0.000,C 90.000,E1 18.109} C_DIS
LIN {X 0.095,Y -395.818,Z 938.887,A 0.000,B 0.000,C 90.000,E1 15.607} C_DIS
LIN {X -0.168,Y -399.570,Z 938.871,A 0.000,B 0.000,C 90.000,E1 12.827} C_DIS
LIN {X -0.101,Y -403.822,Z 938.856,A 0.000,B 0.000,C 90.000,E1 10.018} C_DIS
LIN {X -0.115,Y -408.000,Z 938.842,A 0.000,B 0.000,C 90.000,E1 7.587} C_DIS
LIN {X -0.041,Y -414.556,Z 938.823,A 0.000,B 0.000,C 90.000,E1 4.131} C_DIS
LIN {X -0.166,Y -422.852,Z 938.802,A 0.000,B 0.000,C 90.000,E1 0.401} C_DIS
LIN {X -0.165,Y -425.974,Z 938.795,A 0.000,B 0.000,C 90.000,E1 359.141} C_DIS
LIN {X -0.024,Y -428.655,Z 938.790,A 0.000,B 0.000,C 90.000,E1 358.282} C_DIS
LIN {X 0.088,Y -430.948,Z 938.788,A 0.000,B 0.000,C 90.000,E1 357.764} C_DIS
LIN {X 0.007,Y -435.325,Z 938.784,A 0.000,B 0.000,C 90.000,E1 357.192} C_DIS
LIN {X -0.190,Y -436.110,Z 938.784,A 0.000,B 0.000,C 90.000,E1 357.135} C_DIS
LIN {X 0.007,Y -440.471,Z 938.782,A 0.000,B 0.000,C 90.000,E1 356.788} C_DIS
LIN {X 0.177,Y -446.406,Z 938.780,A 0.000,B 0.000,C 90.000,E1 356.445} C_DIS
LIN {X 0.048,Y -456.396,Z 938.778,A 0.000,B 0.000,C 90.000,E1 355.988} C_DIS
LIN {X 0.026,Y -469.859,Z 938.774,A 0.000,B 0.000,C 90.000,E1 355.298} C_DIS
LIN {X -0.235,Y -481.552,Z 938.771,A 0.000,B 0.000,C 90.000,E1 354.723} C_DIS
LIN {X 0.131,Y -491.605,Z 938.768,A 0.000,B 0.000,C 90.000,E1 354.147} C_DIS
LIN {X 0.033,Y -506.089,Z 938.763,A 0.000,B 0.000,C 90.000,E1 353.337} C_DIS
LIN {X -0.144,Y -514.049,Z 938.760,A 0.000,B 0.000,C 90.000,E1 352.875} C_DIS
LIN {X -0.058,Y -521.992,Z 938.758,A 0.000,B 0.000,C 90.000,E1 352.356} C_DIS
LIN {X -0.252,Y -529.589,Z 938.755,A 0.000,B 0.000,C 90.000,E1 351.837} C_DIS
LIN {X -0.035,Y -536.893,Z 938.751,A 0.000,B 0.000,C 90.000,E1 351.254} C_DIS
LIN {X -0.116,Y -542.577,Z 938.749,A 0.000,B 0.000,C 90.000,E1 350.792} C_DIS
LIN {X 0.117,Y -549.394,Z 938.745,A 0.000,B 0.000,C 90.000,E1 350.151} C_DIS
LIN {X -0.026,Y -555.883,Z 938.742,A 0.000,B 0.000,C 90.000,E1 349.511} C_DIS
LIN {X 0.056,Y -561.842,Z 938.738,A 0.000,B 0.000,C 90.000,E1 348.814} C_DIS
LIN {X -0.016,Y -568.581,Z 938.733,A 0.000,B 0.000,C 90.000,E1 347.993} C_DIS
LIN {X -0.086,Y -571.673,Z 938.731,A 0.000,B 0.000,C 90.000,E1 347.589} C_DIS
LIN {X -0.172,Y -578.403,Z 938.726,A 0.000,B 0.000,C 90.000,E1 346.645} C_DIS
LIN {X 0.163,Y -582.790,Z 938.722,A 0.000,B 0.000,C 90.000,E1 345.936} C_DIS
LIN {X 0.216,Y -588.568,Z 938.717,A 0.000,B 0.000,C 90.000,E1 344.991} C_DIS
LIN {X -0.001,Y -593.019,Z 938.712,A 0.000,B 0.000,C 90.000,E1 344.212} C_DIS
LIN {X 0.170,Y -597.986,Z 938.707,A 0.000,B 0.000,C 90.000,E1 343.268} C_DIS
LIN {X -0.053,Y -603.093,Z 938.701,A 0.000,B 0.000,C 90.000,E1 342.236} C_DIS
LIN {X 0.180,Y -608.131,Z 938.695,A 0.000,B 0.000,C 90.000,E1 341.167} C_DIS
LIN {X 0.063,Y -613.445,Z 938.689,A 0.000,B 0.000,C 90.000,E1 340.007} C_DIS
LIN {X 0.260,Y -617.851,Z 938.683,A 0.000,B 0.000,C 90.000,E1 338.954} C_DIS
LIN {X 0.284,Y -622.901,Z 938.676,A 0.000,B 0.000,C 90.000,E1 337.667} C_DIS
LIN {X 0.036,Y -625.727,Z 938.672,A 0.000,B 0.000,C 90.000,E1 336.922} C_DIS
LIN {X -0.170,Y -629.294,Z 938.666,A 0.000,B 0.000,C 90.000,E1 335.921} C_DIS
LIN {X -0.097,Y -631.866,Z 938.662,A 0.000,B 0.000,C 90.000,E1 335.153} C_DIS
LIN {X -0.226,Y -635.141,Z 938.656,A 0.000,B 0.000,C 90.000,E1 334.152} C_DIS
LIN {X 0.013,Y -638.834,Z 938.649,A 0.000,B 0.000,C 90.000,E1 332.871} C_DIS
LIN {X 0.185,Y -640.893,Z 938.645,A 0.000,B 0.000,C 90.000,E1 332.103} C_DIS
LIN {X -0.123,Y -643.484,Z 938.640,A 0.000,B 0.000,C 90.000,E1 331.129} C_DIS
LIN {X 0.067,Y -647.011,Z 938.631,A 0.000,B 0.000,C 90.000,E1 329.616} C_DIS
LIN {X -0.319,Y -649.571,Z 938.624,A 0.000,B 0.000,C 90.000,E1 328.408} C_DIS
LIN {X -0.282,Y -650.952,Z 938.620,A 0.000,B 0.000,C 90.000,E1 327.661} C_DIS
LIN {X -0.232,Y -652.198,Z 938.616,A 0.000,B 0.000,C 90.000,E1 326.914} C_DIS
LIN {X -0.183,Y -653.984,Z 938.609,A 0.000,B 0.000,C 90.000,E1 325.674} C_DIS
LIN {X 0.268,Y -655.512,Z 938.602,A 0.000,B 0.000,C 90.000,E1 324.402} C_DIS
LIN {X 0.284,Y -656.598,Z 938.597,A 0.000,B 0.000,C 90.000,E1 323.417} C_DIS
LIN {X -0.200,Y -657.869,Z 938.589,A 0.000,B 0.000,C 90.000,E1 321.984} C_DIS
LIN {X 0.174,Y -659.411,Z 938.578,A 0.000,B 0.000,C 90.000,E1 319.989} C_DIS
LIN {X 0.069,Y -660.520,Z 938.570,A 0.000,B 0.000,C 90.000,E1 318.528} C_DIS
LIN {X -0.007,Y -661.717,Z 938.562,A 0.000,B 0.000,C 90.000,E1 317.067} C_DIS
LIN {X 0.386,Y -662.904,Z 938.553,A 0.000,B 0.000,C 90.000,E1 315.567} C_DIS
LIN {X -0.161,Y -664.995,Z 938.540,A 0.000,B 0.000,C 90.000,E1 313.176} C_DIS
LIN {X 0.296,Y -666.384,Z 938.532,A 0.000,B 0.000,C 90.000,E1 311.676} C_DIS
LIN {X -0.108,Y -667.728,Z 938.524,A 0.000,B 0.000,C 90.000,E1 310.253} C_DIS
LIN {X -0.055,Y -668.810,Z 938.517,A 0.000,B 0.000,C 90.000,E1 309.036} C_DIS
LIN {X 0.110,Y -669.770,Z 938.510,A 0.000,B 0.000,C 90.000,E1 307.810} C_DIS
LIN {X -0.225,Y -670.382,Z 938.505,A 0.000,B 0.000,C 90.000,E1 306.870} C_DIS
LIN {X -0.015,Y -670.765,Z 938.499,A 0.000,B 0.000,C 90.000,E1 305.884} C_DIS
LIN {X -0.101,Y -671.287,Z 938.490,A 0.000,B 0.000,C 90.000,E1 304.199} C_DIS
LIN {X 0.012,Y -672.072,Z 938.481,A 0.000,B 0.000,C 90.000,E1 302.498} C_DIS
LIN {X 0.385,Y -672.729,Z 938.474,A 0.000,B 0.000,C 90.000,E1 301.258} C_DIS
LIN {X -0.002,Y -676.465,Z 938.452,A 0.000,B 0.000,C 90.000,E1 297.436} C_DIS
LIN {X -0.288,Y -679.558,Z 938.442,A 0.000,B 0.000,C 90.000,E1 295.540} C_DIS
LIN {X -0.191,Y -681.474,Z 938.435,A 0.000,B 0.000,C 90.000,E1 294.335} C_DIS
LIN {X -0.279,Y -682.760,Z 938.430,A 0.000,B 0.000,C 90.000,E1 293.387} C_DIS
LIN {X -0.139,Y -683.234,Z 938.427,A 0.000,B 0.000,C 90.000,E1 292.898} C_DIS
LIN {X 0.066,Y -683.360,Z 938.426,A 0.000,B 0.000,C 90.000,E1 292.642} C_DIS
LIN {X 0.010,Y -683.288,Z 938.425,A 0.000,B 0.000,C 90.000,E1 292.408} C_DIS
LIN {X -0.216,Y -682.718,Z 938.422,A 0.000,B 0.000,C 90.000,E1 291.950} C_DIS
LIN {X -0.269,Y -681.962,Z 938.421,A 0.000,B 0.000,C 90.000,E1 291.716} C_DIS
LIN {X -0.223,Y -679.888,Z 938.419,A 0.000,B 0.000,C 90.000,E1 291.354} C_DIS
LIN {X -0.033,Y -678.022,Z 938.417,A 0.000,B 0.000,C 90.000,E1 291.099} C_DIS
LIN {X 0.059,Y -676.773,Z 938.417,A 0.000,B 0.000,C 90.000,E1 290.972} C_DIS
LIN {X -0.035,Y -670.278,Z 938.414,A 0.000,B 0.000,C 90.000,E1 290.556} C_DIS
LIN {X 0.277,Y -664.342,Z 938.412,A 0.000,B 0.000,C 90.000,E1 290.174} C_DIS
LIN {X 0.190,Y -662.054,Z 938.411,A 0.000,B 0.000,C 90.000,E1 289.993} C_DIS
LIN {X 0.150,Y -662.034,Z 938.411,A 0.000,B 0.000,C 90.000,E1 289.993} C_DIS
LIN {X -0.190,Y -661.536,Z 938.410,A 0.000,B 0.000,C 90.000,E1 289.866} C_DIS
LIN {X 0.164,Y -662.012,Z 938.409,A 0.000,B 0.000,C 90.000,E1 289.504} C_DIS
LIN {X 0.008,Y -663.791,Z 938.406,A 0.000,B 0.000,C 90.000,E1 289.033} C_DIS
LIN {X -0.215,Y -670.538,Z 938.399,A 0.000,B 0.000,C 90.000,E1 287.764} C_DIS
LIN {X -0.226,Y -674.042,Z 938.395,A 0.000,B 0.000,C 90.000,E1 287.040} C_DIS
LIN {X -0.153,Y -676.102,Z 938.392,A 0.000,B 0.000,C 90.000,E1 286.551} C_DIS
LIN {X -0.310,Y -678.651,Z 938.388,A 0.000,B 0.000,C 90.000,E1 285.843} C_DIS
LIN {X 0.222,Y -680.688,Z 938.384,A 0.000,B 0.000,C 90.000,E1 285.079} C_DIS
LIN {X 0.326,Y -681.808,Z 938.381,A 0.000,B 0.000,C 90.000,E1 284.592} C_DIS
LIN {X 0.203,Y -683.706,Z 938.376,A 0.000,B 0.000,C 90.000,E1 283.647} C_DIS
LIN {X 0.125,Y -684.877,Z 938.372,A 0.000,B 0.000,C 90.000,E1 282.939} C_DIS
LIN {X -0.112,Y -686.025,Z 938.367,A 0.000,B 0.000,C 90.000,E1 282.007} C_DIS
LIN {X -0.132,Y -686.264,Z 938.365,A 0.000,B 0.000,C 90.000,E1 281.771} C_DIS
LIN {X -0.174,Y -686.471,Z 938.363,A 0.000,B 0.000,C 90.000,E1 281.299} C_DIS
LIN {X -0.346,Y -686.458,Z 938.360,A 0.000,B 0.000,C 90.000,E1 280.838} C_DIS
LIN {X 0.286,Y -686.143,Z 938.357,A 0.000,B 0.000,C 90.000,E1 280.310} C_DIS
LIN {X 0.262,Y -685.925,Z 938.356,A 0.000,B 0.000,C 90.000,E1 280.074} C_DIS
LIN {X 0.094,Y -685.020,Z 938.354,A 0.000,B 0.000,C 90.000,E1 279.613} C_DIS
LIN {X -0.076,Y -683.750,Z 938.351,A 0.000,B 0.000,C 90.000,E1 279.151} C_DIS
LIN {X -0.146,Y -682.124,Z 938.348,A 0.000,B 0.000,C 90.000,E1 278.681} C_DIS
LIN {X -0.288,Y -681.211,Z 938.347,A 0.000,B 0.000,C 90.000,E1 278.454} C_DIS
LIN {X 0.146,Y -677.840,Z 938.343,A 0.000,B 0.000,C 90.000,E1 277.701} C_DIS
LIN {X -0.282,Y -672.917,Z 938.338,A 0.000,B 0.000,C 90.000,E1 276.777} C_DIS
LIN {X 0.144,Y -670.240,Z 938.335,A 0.000,B 0.000,C 90.000,E1 276.258} C_DIS
LIN {X -0.116,Y -667.274,Z 938.332,A 0.000,B 0.000,C 90.000,E1 275.796} C_DIS
LIN {X 0.268,Y -663.972,Z 938.329,A 0.000,B 0.000,C 90.000,E1 275.277} C_DIS
LIN {X -0.128,Y -659.159,Z 938.326,A 0.000,B 0.000,C 90.000,E1 274.702} C_DIS
LIN {X 0.146,Y -654.955,Z 938.323,A 0.000,B 0.000,C 90.000,E1 274.188} C_DIS
LIN {X -0.314,Y -649.150,Z 938.320,A 0.000,B 0.000,C 90.000,E1 273.612} C_DIS
LIN {X 0.026,Y -644.247,Z 938.317,A 0.000,B 0.000,C 90.000,E1 273.094} C_DIS
LIN {X -0.170,Y -637.613,Z 938.314,A 0.000,B 0.000,C 90.000,E1 272.522} C_DIS
LIN {X 0.010,Y -630.678,Z 938.311,A 0.000,B 0.000,C 90.000,E1 271.949} C_DIS
LIN {X -0.066,Y -623.138,Z 938.308,A 0.000,B 0.000,C 90.000,E1 271.432} C_DIS
LIN {X -0.015,Y -617.023,Z 938.306,A 0.000,B 0.000,C 90.000,E1 271.031} C_DIS
LIN {X -0.285,Y -610.921,Z 938.304,A 0.000,B 0.000,C 90.000,E1 270.688} C_DIS
LIN {X -0.059,Y -602.658,Z 938.301,A 0.000,B 0.000,C 90.000,E1 270.229} C_DIS
LIN {X -0.214,Y -597.669,Z 938.300,A 0.000,B 0.000,C 90.000,E1 270.000} C_DIS
LIN {X -0.277,Y -590.723,Z 938.298,A 0.000,B 0.000,C 90.000,E1 269.714} C_DIS
LIN {X 0.024,Y -585.379,Z 938.297,A 0.000,B 0.000,C 90.000,E1 269.484} C_DIS
LIN {X -0.004,Y -577.740,Z 938.296,A 0.000,B 0.000,C 90.000,E1 269.255} C_DIS
LIN {X 0.234,Y -571.657,Z 938.295,A 0.000,B 0.000,C 90.000,E1 269.083} C_DIS
LIN {X -0.064,Y -563.555,Z 938.294,A 0.000,B 0.000,C 90.000,E1 268.969} C_DIS
LIN {X -0.186,Y -557.469,Z 938.294,A 0.000,B 0.000,C 90.000,E1 268.912} C_DIS
LIN {X 0.248,Y -554.318,Z 938.294,A 0.000,B 0.000,C 90.000,E1 268.854} C_DIS
LIN {X -0.018,Y -551.242,Z 938.294,A 0.000,B 0.000,C 90.000,E1 268.854} C_DIS
LIN {X 0.270,Y -549.705,Z 938.294,A 0.000,B 0.000,C 90.000,E1 268.797} C_DIS
LIN {X 0.231,Y -549.515,Z 938.294,A 0.000,B 0.000,C 90.000,E1 268.797} C_DIS
LIN {X -0.050,Y -547.936,Z 938.292,A 0.000,B 0.000,C 90.000,E1 268.625} C_DIS
LIN {X -0.001,Y -545.496,Z 938.291,A 0.000,B 0.000,C 90.000,E1 268.339} C_DIS
LIN {X 0.253,Y -544.066,Z 938.290,A 0.000,B 0.000,C 90.000,E1 268.167} C_DIS
LIN {X 0.213,Y -544.057,Z 938.290,A 0.000,B 0.000,C 90.000,E1 268.167} C_DIS
LIN {X 0.208,Y -543.251,Z 938.288,A 0.000,B 0.000,C 90.000,E1 267.764} C_DIS
LIN {X -0.191,Y -540.214,Z 938.268,A 0.000,B 0.000,C 90.000,E1 264.261} C_DIS
LIN {X 0.063,Y -538.864,Z 938.257,A 0.000,B 0.000,C 90.000,E1 262.243} C_DIS
LIN {X 0.241,Y -538.048,Z 938.251,A 0.000,B 0.000,C 90.000,E1 261.084} C_DIS
LIN {X -0.185,Y -537.236,Z 938.246,A 0.000,B 0.000,C 90.000,E1 260.274} C_DIS
LIN {X -0.062,Y -536.533,Z 938.243,A 0.000,B 0.000,C 90.000,E1 259.690} C_DIS
LIN {X 0.174,Y -534.891,Z 938.236,A 0.000,B 0.000,C 90.000,E1 258.522} C_DIS
LIN {X -0.265,Y -531.232,Z 938.220,A 0.000,B 0.000,C 90.000,E1 255.700} C_DIS
LIN {X 0.206,Y -529.210,Z 938.211,A 0.000,B 0.000,C 90.000,E1 253.921} C_DIS
LIN {X 0.268,Y -527.163,Z 938.201,A 0.000,B 0.000,C 90.000,E1 252.181} C_DIS
LIN {X -0.044,Y -524.948,Z 938.192,A 0.000,B 0.000,C 90.000,E1 250.477} C_DIS
LIN {X 0.087,Y -522.725,Z 938.182,A 0.000,B 0.000,C 90.000,E1 248.720} C_DIS
LIN {X 0.233,Y -521.210,Z 938.175,A 0.000,B 0.000,C 90.000,E1 247.539} C_DIS
LIN {X 0.172,Y -518.627,Z 938.166,A 0.000,B 0.000,C 90.000,E1 245.793} C_DIS
LIN {X 0.134,Y -516.283,Z 938.158,A 0.000,B 0.000,C 90.000,E1 244.332} C_DIS
LIN {X 0.046,Y -514.921,Z 938.153,A 0.000,B 0.000,C 90.000,E1 243.461} C_DIS
LIN {X 0.164,Y -512.555,Z 938.144,A 0.000,B 0.000,C 90.000,E1 241.975} C_DIS
LIN {X 0.038,Y -510.100,Z 938.136,A 0.000,B 0.000,C 90.000,E1 240.511} C_DIS
LIN {X -0.013,Y -508.009,Z 938.130,A 0.000,B 0.000,C 90.000,E1 239.331} C_DIS
LIN {X 0.160,Y -505.692,Z 938.123,A 0.000,B 0.000,C 90.000,E1 238.122} C_DIS
LIN {X -0.016,Y -503.822,Z 938.118,A 0.000,B 0.000,C 90.000,E1 237.248} C_DIS
LIN {X -0.162,Y -499.710,Z 938.108,A 0.000,B 0.000,C 90.000,E1 235.468} C_DIS
LIN {X 0.033,Y -494.910,Z 938.096,A 0.000,B 0.000,C 90.000,E1 233.336} C_DIS
LIN {X 0.013,Y -491.669,Z 938.088,A 0.000,B 0.000,C 90.000,E1 231.823} C_DIS
LIN {X 0.234,Y -488.299,Z 938.080,A 0.000,B 0.000,C 90.000,E1 230.275} C_DIS
LIN {X -0.029,Y -483.395,Z 938.068,A 0.000,B 0.000,C 90.000,E1 228.162} C_DIS
LIN {X 0.222,Y -478.536,Z 938.056,A 0.000,B 0.000,C 90.000,E1 225.972} C_DIS
LIN {X 0.225,Y -474.420,Z 938.045,A 0.000,B 0.000,C 90.000,E1 224.109} C_DIS
LIN {X -0.053,Y -471.646,Z 938.038,A 0.000,B 0.000,C 90.000,E1 222.894} C_DIS
LIN {X 0.081,Y -468.215,Z 938.030,A 0.000,B 0.000,C 90.000,E1 221.310} C_DIS
LIN {X -0.284,Y -462.689,Z 938.016,A 0.000,B 0.000,C 90.000,E1 218.830} C_DIS
LIN {X -0.248,Y -459.258,Z 938.007,A 0.000,B 0.000,C 90.000,E1 217.237} C_DIS
LIN {X 0.088,Y -455.805,Z 937.998,A 0.000,B 0.000,C 90.000,E1 215.598} C_DIS
LIN {X 0.089,Y -452.315,Z 937.989,A 0.000,B 0.000,C 90.000,E1 213.992} C_DIS
LIN {X -0.229,Y -448.685,Z 937.980,A 0.000,B 0.000,C 90.000,E1 212.418} C_DIS
LIN {X -0.172,Y -444.414,Z 937.969,A 0.000,B 0.000,C 90.000,E1 210.463} C_DIS
LIN {X -0.063,Y -440.144,Z 937.958,A 0.000,B 0.000,C 90.000,E1 208.487} C_DIS
LIN {X 0.099,Y -436.658,Z 937.949,A 0.000,B 0.000,C 90.000,E1 206.821} C_DIS
LIN {X 0.012,Y -432.230,Z 937.938,A 0.000,B 0.000,C 90.000,E1 204.847} C_DIS
LIN {X -0.168,Y -428.570,Z 937.929,A 0.000,B 0.000,C 90.000,E1 203.206} C_DIS
LIN {X -0.197,Y -424.872,Z 937.920,A 0.000,B 0.000,C 90.000,E1 201.535} C_DIS
LIN {X -0.129,Y -420.459,Z 937.908,A 0.000,B 0.000,C 90.000,E1 199.504} C_DIS
LIN {X 0.102,Y -415.692,Z 937.895,A 0.000,B 0.000,C 90.000,E1 197.094} C_DIS
LIN {X -0.196,Y -412.281,Z 937.886,A 0.000,B 0.000,C 90.000,E1 195.426} C_DIS
LIN {X 0.112,Y -409.436,Z 937.878,A 0.000,B 0.000,C 90.000,E1 194.008} C_DIS
LIN {X 0.095,Y -403.922,Z 937.863,A 0.000,B 0.000,C 90.000,E1 191.243} C_DIS
LIN {X 0.086,Y -399.924,Z 937.851,A 0.000,B 0.000,C 90.000,E1 189.151} C_DIS
LIN {X 0.001,Y -396.529,Z 937.841,A 0.000,B 0.000,C 90.000,E1 187.409} C_DIS
LIN {X -0.174,Y -393.749,Z 937.833,A 0.000,B 0.000,C 90.000,E1 186.024} C_DIS
LIN {X -0.126,Y -390.473,Z 937.824,A 0.000,B 0.000,C 90.000,E1 184.245} C_DIS
LIN {X 0.070,Y -386.163,Z 937.810,A 0.000,B 0.000,C 90.000,E1 181.718} C_DIS
LIN {X -0.059,Y -383.592,Z 937.800,A 0.000,B 0.000,C 90.000,E1 179.943} C_DIS
LIN {X -0.007,Y -382.544,Z 937.794,A 0.000,B 0.000,C 90.000,E1 178.854} C_DIS
LIN {X -0.122,Y -382.303,Z 937.792,A 0.000,B 0.000,C 90.000,E1 178.511} C_DIS
LIN {X 0.042,Y -382.242,Z 937.788,A 0.000,B 0.000,C 90.000,E1 177.764} C_DIS
LIN {X -0.194,Y -382.617,Z 937.784,A 0.000,B 0.000,C 90.000,E1 177.078} C_DIS
LIN {X 0.091,Y -383.017,Z 937.782,A 0.000,B 0.000,C 90.000,E1 176.674} C_DIS
LIN {X -0.027,Y -383.833,Z 937.780,A 0.000,B 0.000,C 90.000,E1 176.331} C_DIS
LIN {X -0.144,Y -384.793,Z 937.778,A 0.000,B 0.000,C 90.000,E1 175.988} C_DIS
LIN {X 0.152,Y -386.254,Z 937.776,A 0.000,B 0.000,C 90.000,E1 175.584} C_DIS
LIN {X 0.041,Y -388.163,Z 937.774,A 0.000,B 0.000,C 90.000,E1 175.241} C_DIS
LIN {X 0.027,Y -389.239,Z 937.773,A 0.000,B 0.000,C 90.000,E1 175.065} C_DIS
LIN {X 0.045,Y -395.426,Z 937.768,A 0.000,B 0.000,C 90.000,E1 174.318} C_DIS
LIN {X 0.081,Y -402.599,Z 937.765,A 0.000,B 0.000,C 90.000,E1 173.685} C_DIS
LIN {X 0.073,Y -421.475,Z 937.757,A 0.000,B 0.000,C 90.000,E1 172.186} C_DIS
LIN {X -0.067,Y -432.350,Z 937.752,A 0.000,B 0.000,C 90.000,E1 171.310} C_DIS
LIN {X 0.185,Y -441.600,Z 937.747,A 0.000,B 0.000,C 90.000,E1 170.500} C_DIS
LIN {X 0.155,Y -450.583,Z 937.743,A 0.000,B 0.000,C 90.000,E1 169.690} C_DIS
LIN {X 0.085,Y -459.208,Z 937.738,A 0.000,B 0.000,C 90.000,E1 168.870} C_DIS
LIN {X -0.198,Y -465.055,Z 937.735,A 0.000,B 0.000,C 90.000,E1 168.342} C_DIS
LIN {X -0.005,Y -471.790,Z 937.731,A 0.000,B 0.000,C 90.000,E1 167.589} C_DIS
LIN {X 0.067,Y -478.390,Z 937.727,A 0.000,B 0.000,C 90.000,E1 166.825} C_DIS
LIN {X 0.050,Y -485.890,Z 937.722,A 0.000,B 0.000,C 90.000,E1 165.936} C_DIS
LIN {X 0.074,Y -491.997,Z 937.718,A 0.000,B 0.000,C 90.000,E1 165.172} C_DIS
LIN {X -0.014,Y -496.655,Z 937.714,A 0.000,B 0.000,C 90.000,E1 164.574} C_DIS
LIN {X -0.084,Y -505.254,Z 937.708,A 0.000,B 0.000,C 90.000,E1 163.378} C_DIS
LIN {X -0.028,Y -513.358,Z 937.701,A 0.000,B 0.000,C 90.000,E1 162.181} C_DIS
LIN {X -0.032,Y -518.128,Z 937.697,A 0.000,B 0.000,C 90.000,E1 161.456} C_DIS
LIN {X -0.243,Y -521.062,Z 937.695,A 0.000,B 0.000,C 90.000,E1 161.040} C_DIS
LIN {X 0.047,Y -529.355,Z 937.687,A 0.000,B 0.000,C 90.000,E1 159.699} C_DIS
LIN {X -0.224,Y -535.806,Z 937.682,A 0.000,B 0.000,C 90.000,E1 158.720} C_DIS
LIN {X -0.081,Y -541.044,Z 937.677,A 0.000,B 0.000,C 90.000,E1 157.847} C_DIS
LIN {X -0.213,Y -550.305,Z 937.668,A 0.000,B 0.000,C 90.000,E1 156.305} C_DIS
LIN {X 0.091,Y -555.142,Z 937.664,A 0.000,B 0.000,C 90.000,E1 155.433} C_DIS
LIN {X -0.027,Y -561.180,Z 937.657,A 0.000,B 0.000,C 90.000,E1 154.332} C_DIS
LIN {X -0.014,Y -564.761,Z 937.654,A 0.000,B 0.000,C 90.000,E1 153.640} C_DIS
LIN {X -0.066,Y -568.935,Z 937.649,A 0.000,B 0.000,C 90.000,E1 152.820} C_DIS
LIN {X -0.065,Y -574.654,Z 937.642,A 0.000,B 0.000,C 90.000,E1 151.591} C_DIS
LIN {X -0.124,Y -579.524,Z 937.636,A 0.000,B 0.000,C 90.000,E1 150.511} C_DIS
LIN {X -0.034,Y -585.176,Z 937.629,A 0.000,B 0.000,C 90.000,E1 149.154} C_DIS
LIN {X 0.182,Y -588.369,Z 937.624,A 0.000,B 0.000,C 90.000,E1 148.329} C_DIS
LIN {X -0.291,Y -593.469,Z 937.617,A 0.000,B 0.000,C 90.000,E1 147.041} C_DIS
LIN {X -0.085,Y -597.504,Z 937.611,A 0.000,B 0.000,C 90.000,E1 145.960} C_DIS
LIN {X 0.162,Y -603.254,Z 937.602,A 0.000,B 0.000,C 90.000,E1 144.356} C_DIS
LIN {X -0.177,Y -609.658,Z 937.592,A 0.000,B 0.000,C 90.000,E1 142.557} C_DIS
LIN {X 0.198,Y -615.227,Z 937.583,A 0.000,B 0.000,C 90.000,E1 140.964} C_DIS
LIN {X -0.108,Y -619.947,Z 937.576,A 0.000,B 0.000,C 90.000,E1 139.703} C_DIS
LIN {X -0.076,Y -625.562,Z 937.568,A 0.000,B 0.000,C 90.000,E1 138.162} C_DIS
LIN {X 0.198,Y -630.449,Z 937.560,A 0.000,B 0.000,C 90.000,E1 136.863} C_DIS
LIN {X -0.153,Y -633.514,Z 937.556,A 0.000,B 0.000,C 90.000,E1 136.134} C_DIS
LIN {X 0.140,Y -639.266,Z 937.548,A 0.000,B 0.000,C 90.000,E1 134.595} C_DIS
LIN {X -0.285,Y -644.044,Z 937.541,A 0.000,B 0.000,C 90.000,E1 133.380} C_DIS
LIN {X 0.186,Y -650.736,Z 937.531,A 0.000,B 0.000,C 90.000,E1 131.595} C_DIS
LIN {X -0.074,Y -656.417,Z 937.523,A 0.000,B 0.000,C 90.000,E1 130.135} C_DIS
LIN {X 0.336,Y -662.959,Z 937.513,A 0.000,B 0.000,C 90.000,E1 128.382} C_DIS
LIN {X -0.080,Y -666.653,Z 937.508,A 0.000,B 0.000,C 90.000,E1 127.443} C_DIS
LIN {X -0.357,Y -672.044,Z 937.500,A 0.000,B 0.000,C 90.000,E1 126.011} C_DIS
LIN {X 0.286,Y -674.627,Z 937.496,A 0.000,B 0.000,C 90.000,E1 125.231} C_DIS
LIN {X 0.157,Y -678.574,Z 937.489,A 0.000,B 0.000,C 90.000,E1 124.040} C_DIS
LIN {X -0.459,Y -680.834,Z 937.485,A 0.000,B 0.000,C 90.000,E1 123.372} C_DIS
LIN {X 0.072,Y -684.112,Z 937.479,A 0.000,B 0.000,C 90.000,E1 122.133} C_DIS
LIN {X 0.100,Y -685.849,Z 937.475,A 0.000,B 0.000,C 90.000,E1 121.416} C_DIS
LIN {X 0.132,Y -687.970,Z 937.469,A 0.000,B 0.000,C 90.000,E1 120.463} C_DIS
LIN {X -0.164,Y -689.770,Z 937.464,A 0.000,B 0.000,C 90.000,E1 119.539} C_DIS
LIN {X 0.166,Y -691.280,Z 937.459,A 0.000,B 0.000,C 90.000,E1 118.565} C_DIS
LIN {X -0.094,Y -692.416,Z 937.454,A 0.000,B 0.000,C 90.000,E1 117.641} C_DIS
LIN {X -0.046,Y -693.145,Z 937.448,A 0.000,B 0.000,C 90.000,E1 116.693} C_DIS
LIN {X 0.075,Y -693.434,Z 937.444,A 0.000,B 0.000,C 90.000,E1 115.976} C_DIS
LIN {X 0.143,Y -693.580,Z 937.439,A 0.000,B 0.000,C 90.000,E1 115.027} C_DIS
LIN {X 0.210,Y -693.463,Z 937.434,A 0.000,B 0.000,C 90.000,E1 114.079} C_DIS
LIN {X -0.179,Y -693.350,Z 937.433,A 0.000,B 0.000,C 90.000,E1 113.875} C_DIS
LIN {X 0.028,Y -692.630,Z 937.430,A 0.000,B 0.000,C 90.000,E1 113.387} C_DIS
LIN {X -0.004,Y -691.954,Z 937.429,A 0.000,B 0.000,C 90.000,E1 113.153} C_DIS
LIN {X -0.165,Y -690.000,Z 937.426,A 0.000,B 0.000,C 90.000,E1 112.695} C_DIS
LIN {X -0.314,Y -689.251,Z 937.425,A 0.000,B 0.000,C 90.000,E1 112.589} C_DIS
LIN {X -0.199,Y -688.165,Z 937.425,A 0.000,B 0.000,C 90.000,E1 112.461} C_DIS
LIN {X -0.085,Y -686.890,Z 937.424,A 0.000,B 0.000,C 90.000,E1 112.333} C_DIS
LIN {X -0.351,Y -682.677,Z 937.422,A 0.000,B 0.000,C 90.000,E1 112.025} C_DIS
LIN {X -0.081,Y -680.801,Z 937.422,A 0.000,B 0.000,C 90.000,E1 111.897} C_DIS
LIN {X 0.185,Y -678.050,Z 937.421,A 0.000,B 0.000,C 90.000,E1 111.770} C_DIS
LIN {X 0.055,Y -675.969,Z 937.421,A 0.000,B 0.000,C 90.000,E1 111.716} C_DIS
LIN {X -0.073,Y -673.298,Z 937.420,A 0.000,B 0.000,C 90.000,E1 111.663} C_DIS
LIN {X -0.201,Y -668.638,Z 937.420,A 0.000,B 0.000,C 90.000,E1 111.589} C_DIS
LIN {X 0.174,Y -666.844,Z 937.420,A 0.000,B 0.000,C 90.000,E1 111.535} C_DIS
LIN {X -0.165,Y -660.014,Z 937.420,A 0.000,B 0.000,C 90.000,E1 111.535} C_DIS
LIN {X -0.213,Y -638.341,Z 937.420,A 0.000,B 0.000,C 90.000,E1 111.535} C_DIS
LIN {X 0.207,Y -633.851,Z 937.419,A 0.000,B 0.000,C 90.000,E1 111.461} C_DIS
LIN {X -0.111,Y -628.055,Z 937.419,A 0.000,B 0.000,C 90.000,E1 111.408} C_DIS
LIN {X 0.099,Y -622.639,Z 937.418,A 0.000,B 0.000,C 90.000,E1 111.280} C_DIS
LIN {X -0.035,Y -615.565,Z 937.417,A 0.000,B 0.000,C 90.000,E1 111.099} C_DIS
LIN {X -0.081,Y -608.547,Z 937.416,A 0.000,B 0.000,C 90.000,E1 110.844} C_DIS
LIN {X -0.200,Y -603.122,Z 937.414,A 0.000,B 0.000,C 90.000,E1 110.610} C_DIS
LIN {X -0.032,Y -597.708,Z 937.413,A 0.000,B 0.000,C 90.000,E1 110.301} C_DIS
LIN {X -0.192,Y -591.020,Z 937.410,A 0.000,B 0.000,C 90.000,E1 109.885} C_DIS
LIN {X -0.154,Y -578.092,Z 937.405,A 0.000,B 0.000,C 90.000,E1 108.960} C_DIS
LIN {X 0.034,Y -570.984,Z 937.403,A 0.000,B 0.000,C 90.000,E1 108.544} C_DIS
LIN {X -0.116,Y -565.912,Z 937.402,A 0.000,B 0.000,C 90.000,E1 108.308} C_DIS
LIN {X -0.182,Y -557.284,Z 937.400,A 0.000,B 0.000,C 90.000,E1 107.946} C_DIS
LIN {X 0.002,Y -553.932,Z 937.399,A 0.000,B 0.000,C 90.000,E1 107.764} C_DIS
LIN {X 0.184,Y -552.145,Z 937.398,A 0.000,B 0.000,C 90.000,E1 107.583} C_DIS
LIN {X 0.146,Y -552.106,Z 937.398,A 0.000,B 0.000,C 90.000,E1 107.583} C_DIS
LIN {X -0.051,Y -551.810,Z 937.397,A 0.000,B 0.000,C 90.000,E1 107.402} C_DIS
LIN {X -0.129,Y -552.560,Z 937.385,A 0.000,B 0.000,C 90.000,E1 105.300} C_DIS
LIN {X 0.172,Y -553.353,Z 937.376,A 0.000,B 0.000,C 90.000,E1 103.592} C_DIS
LIN {X -0.038,Y -554.580,Z 937.365,A 0.000,B 0.000,C 90.000,E1 101.658} C_DIS
LIN {X -0.224,Y -556.143,Z 937.354,A 0.000,B 0.000,C 90.000,E1 99.726} C_DIS
LIN {X -0.151,Y -557.514,Z 937.345,A 0.000,B 0.000,C 90.000,E1 98.049} C_DIS
LIN {X -0.245,Y -558.368,Z 937.339,A 0.000,B 0.000,C 90.000,E1 96.947} C_DIS
LIN {X 0.233,Y -559.309,Z 937.331,A 0.000,B 0.000,C 90.000,E1 95.511} C_DIS
LIN {X 0.181,Y -560.112,Z 937.323,A 0.000,B 0.000,C 90.000,E1 94.131} C_DIS
LIN {X 0.137,Y -560.904,Z 937.315,A 0.000,B 0.000,C 90.000,E1 92.751} C_DIS
LIN {X 0.264,Y -561.758,Z 937.305,A 0.000,B 0.000,C 90.000,E1 90.802} C_DIS
LIN {X 0.101,Y -562.127,Z 937.299,A 0.000,B 0.000,C 90.000,E1 89.714} C_DIS
LIN {X -0.059,Y -562.409,Z 937.292,A 0.000,B 0.000,C 90.000,E1 88.625} C_DIS
LIN {X -0.003,Y -562.826,Z 937.283,A 0.000,B 0.000,C 90.000,E1 86.963} C_DIS
LIN {X 0.231,Y -563.139,Z 937.272,A 0.000,B 0.000,C 90.000,E1 85.008} C_DIS
LIN {X -0.171,Y -563.340,Z 937.263,A 0.000,B 0.000,C 90.000,E1 83.394} C_DIS
LIN {X -0.252,Y -563.525,Z 937.257,A 0.000,B 0.000,C 90.000,E1 82.299} C_DIS
LIN {X -0.025,Y -564.012,Z 937.248,A 0.000,B 0.000,C 90.000,E1 80.622} C_DIS
LIN {X -0.094,Y -564.770,Z 937.237,A 0.000,B 0.000,C 90.000,E1 78.701} C_DIS
LIN {X -0.200,Y -565.664,Z 937.228,A 0.000,B 0.000,C 90.000,E1 77.061} C_DIS
LIN {X -0.159,Y -566.694,Z 937.219,A 0.000,B 0.000,C 90.000,E1 75.408} C_DIS
LIN {X 0.053,Y -567.666,Z 937.210,A 0.000,B 0.000,C 90.000,E1 73.740} C_DIS
LIN {X -0.259,Y -568.592,Z 937.201,A 0.000,B 0.000,C 90.000,E1 72.127} C_DIS
LIN {X 0.341,Y -569.394,Z 937.191,A 0.000,B 0.000,C 90.000,E1 70.423} C_DIS
LIN {X -0.268,Y -569.789,Z 937.185,A 0.000,B 0.000,C 90.000,E1 69.390} C_DIS
LIN {X -0.141,Y -570.135,Z 937.179,A 0.000,B 0.000,C 90.000,E1 68.284} C_DIS
LIN {X -0.009,Y -570.568,Z 937.169,A 0.000,B 0.000,C 90.000,E1 66.357} C_DIS
LIN {X 0.013,Y -570.885,Z 937.160,A 0.000,B 0.000,C 90.000,E1 64.717} C_DIS
LIN {X 0.199,Y -571.100,Z 937.152,A 0.000,B 0.000,C 90.000,E1 63.332} C_DIS
LIN {X 0.128,Y -571.195,Z 937.144,A 0.000,B 0.000,C 90.000,E1 61.975} C_DIS
LIN {X 0.164,Y -571.141,Z 937.135,A 0.000,B 0.000,C 90.000,E1 60.333} C_DIS
LIN {X -0.120,Y -571.228,Z 937.128,A 0.000,B 0.000,C 90.000,E1 58.997} C_DIS
LIN {X -0.349,Y -571.158,Z 937.123,A 0.000,B 0.000,C 90.000,E1 58.201} C_DIS
LIN {X 0.146,Y -570.784,Z 937.116,A 0.000,B 0.000,C 90.000,E1 56.786} C_DIS
LIN {X -0.260,Y -570.544,Z 937.111,A 0.000,B 0.000,C 90.000,E1 56.008} C_DIS
LIN {X 0.068,Y -569.872,Z 937.103,A 0.000,B 0.000,C 90.000,E1 54.609} C_DIS
LIN {X -0.079,Y -569.030,Z 937.096,A 0.000,B 0.000,C 90.000,E1 53.256} C_DIS
LIN {X 0.081,Y -568.021,Z 937.090,A 0.000,B 0.000,C 90.000,E1 52.145} C_DIS
LIN {X 0.116,Y -566.821,Z 937.084,A 0.000,B 0.000,C 90.000,E1 51.045} C_DIS
LIN {X -0.302,Y -565.376,Z 937.078,A 0.000,B 0.000,C 90.000,E1 49.989} C_DIS
LIN {X 0.280,Y -564.601,Z 937.075,A 0.000,B 0.000,C 90.000,E1 49.380} C_DIS
LIN {X 0.161,Y -563.224,Z 937.070,A 0.000,B 0.000,C 90.000,E1 48.566} C_DIS
LIN {X 0.069,Y -560.984,Z 937.064,A 0.000,B 0.000,C 90.000,E1 47.472} C_DIS
LIN {X 0.205,Y -559.806,Z 937.061,A 0.000,B 0.000,C 90.000,E1 46.905} C_DIS
LIN {X 0.002,Y -557.700,Z 937.056,A 0.000,B 0.000,C 90.000,E1 46.095} C_DIS
LIN {X -0.269,Y -556.216,Z 937.053,A 0.000,B 0.000,C 90.000,E1 45.567} C_DIS
LIN {X 0.277,Y -553.698,Z 937.048,A 0.000,B 0.000,C 90.000,E1 44.676} C_DIS
LIN {X 0.363,Y -551.856,Z 937.045,A 0.000,B 0.000,C 90.000,E1 44.109} C_DIS
LIN {X 0.074,Y -548.779,Z 937.041,A 0.000,B 0.000,C 90.000,E1 43.299} C_DIS
LIN {X -0.250,Y -546.586,Z 937.038,A 0.000,B 0.000,C 90.000,E1 42.771} C_DIS
LIN {X -0.023,Y -543.567,Z 937.034,A 0.000,B 0.000,C 90.000,E1 42.043} C_DIS
LIN {X 0.211,Y -540.163,Z 937.030,A 0.000,B 0.000,C 90.000,E1 41.310} C_DIS
LIN {X 0.187,Y -535.722,Z 937.025,A 0.000,B 0.000,C 90.000,E1 40.458} C_DIS
LIN {X -0.057,Y -531.718,Z 937.021,A 0.000,B 0.000,C 90.000,E1 39.769} C_DIS
LIN {X 0.017,Y -523.852,Z 937.014,A 0.000,B 0.000,C 90.000,E1 38.463} C_DIS
LIN {X -0.109,Y -518.147,Z 937.009,A 0.000,B 0.000,C 90.000,E1 37.604} C_DIS
LIN {X 0.014,Y -512.070,Z 937.004,A 0.000,B 0.000,C 90.000,E1 36.710} C_DIS
LIN {X 0.263,Y -507.775,Z 937.001,A 0.000,B 0.000,C 90.000,E1 36.091} C_DIS
LIN {X -0.131,Y -502.107,Z 936.997,A 0.000,B 0.000,C 90.000,E1 35.391} C_DIS
LIN {X -0.156,Y -498.421,Z 936.994,A 0.000,B 0.000,C 90.000,E1 34.945} C_DIS
LIN {X -0.187,Y -491.958,Z 936.990,A 0.000,B 0.000,C 90.000,E1 34.199} C_DIS
LIN {X -0.027,Y -485.043,Z 936.986,A 0.000,B 0.000,C 90.000,E1 33.452} C_DIS
LIN {X 0.220,Y -479.636,Z 936.983,A 0.000,B 0.000,C 90.000,E1 32.880} C_DIS
LIN {X -0.020,Y -471.028,Z 936.978,A 0.000,B 0.000,C 90.000,E1 32.084} C_DIS
LIN {X 0.071,Y -460.601,Z 936.973,A 0.000,B 0.000,C 90.000,E1 31.131} C_DIS
LIN {X 0.159,Y -449.912,Z 936.968,A 0.000,B 0.000,C 90.000,E1 30.207} C_DIS
LIN {X -0.078,Y -437.568,Z 936.962,A 0.000,B 0.000,C 90.000,E1 29.205} C_DIS
LIN {X -0.135,Y -413.278,Z 936.950,A 0.000,B 0.000,C 90.000,E1 27.052} C_DIS
LIN {X 0.023,Y -398.834,Z 936.942,A 0.000,B 0.000,C 90.000,E1 25.591} C_DIS
LIN {X -0.001,Y -396.211,Z 936.940,A 0.000,B 0.000,C 90.000,E1 25.283} C_DIS
LIN {X -0.133,Y -393.634,Z 936.939,A 0.000,B 0.000,C 90.000,E1 24.951} C_DIS
LIN {X 0.218,Y -391.464,Z 936.936,A 0.000,B 0.000,C 90.000,E1 24.515} C_DIS
LIN {X -0.031,Y -389.796,Z 936.934,A 0.000,B 0.000,C 90.000,E1 24.027} C_DIS
LIN {X -0.169,Y -389.032,Z 936.930,A 0.000,B 0.000,C 90.000,E1 23.334} C_DIS
LIN {X -0.120,Y -389.284,Z 936.923,A 0.000,B 0.000,C 90.000,E1 22.078} C_DIS
LIN {X 0.119,Y -392.992,Z 936.901,A 0.000,B 0.000,C 90.000,E1 18.127} C_DIS
LIN {X 0.025,Y -395.880,Z 936.887,A 0.000,B 0.000,C 90.000,E1 15.662} C_DIS
LIN {X 0.148,Y -399.626,Z 936.871,A 0.000,B 0.000,C 90.000,E1 12.827} C_DIS
LIN {X -0.179,Y -404.446,Z 936.854,A 0.000,B 0.000,C 90.000,E1 9.726} C_DIS
LIN {X -0.180,Y -408.644,Z 936.840,A 0.000,B 0.000,C 90.000,E1 7.296} C_DIS
LIN {X -0.091,Y -415.253,Z 936.821,A 0.000,B 0.000,C 90.000,E1 3.841} C_DIS
LIN {X -0.209,Y -423.616,Z 936.801,A 0.000,B 0.000,C 90.000,E1 0.115} C_DIS
LIN {X -0.164,Y -426.006,Z 936.795,A 0.000,B 0.000,C 90.000,E1 359.141} C_DIS
LIN {X -0.054,Y -428.052,Z 936.791,A 0.000,B 0.000,C 90.000,E1 358.453} C_DIS
LIN {X 0.021,Y -429.227,Z 936.790,A 0.000,B 0.000,C 90.000,E1 358.108} C_DIS
LIN {X 0.172,Y -430.673,Z 936.788,A 0.000,B 0.000,C 90.000,E1 357.764} C_DIS
LIN {X 0.208,Y -431.681,Z 936.787,A 0.000,B 0.000,C 90.000,E1 357.593} C_DIS
LIN {X 0.129,Y -436.071,Z 936.784,A 0.000,B 0.000,C 90.000,E1 357.020} C_DIS
LIN {X -0.022,Y -441.041,Z 936.782,A 0.000,B 0.000,C 90.000,E1 356.674} C_DIS
LIN {X 0.121,Y -447.195,Z 936.780,A 0.000,B 0.000,C 90.000,E1 356.331} C_DIS
LIN {X 0.102,Y -455.930,Z 936.777,A 0.000,B 0.000,C 90.000,E1 355.927} C_DIS
LIN {X 0.105,Y -469.316,Z 936.774,A 0.000,B 0.000,C 90.000,E1 355.241} C_DIS
LIN {X 0.120,Y -482.653,Z 936.770,A 0.000,B 0.000,C 90.000,E1 354.546} C_DIS
LIN {X -0.023,Y -492.647,Z 936.767,A 0.000,B 0.000,C 90.000,E1 354.033} C_DIS
LIN {X -0.112,Y -504.144,Z 936.763,A 0.000,B 0.000,C 90.000,E1 353.394} C_DIS
LIN {X -0.094,Y -513.720,Z 936.760,A 0.000,B 0.000,C 90.000,E1 352.818} C_DIS
LIN {X 0.074,Y -521.571,Z 936.757,A 0.000,B 0.000,C 90.000,E1 352.299} C_DIS
LIN {X -0.071,Y -529.149,Z 936.754,A 0.000,B 0.000,C 90.000,E1 351.781} C_DIS
LIN {X 0.091,Y -536.569,Z 936.751,A 0.000,B 0.000,C 90.000,E1 351.197} C_DIS
LIN {X -0.052,Y -543.665,Z 936.748,A 0.000,B 0.000,C 90.000,E1 350.622} C_DIS
LIN {X 0.063,Y -550.496,Z 936.744,A 0.000,B 0.000,C 90.000,E1 349.982} C_DIS
LIN {X 0.083,Y -555.659,Z 936.742,A 0.000,B 0.000,C 90.000,E1 349.454} C_DIS
LIN {X -0.059,Y -561.381,Z 936.738,A 0.000,B 0.000,C 90.000,E1 348.814} C_DIS
LIN {X -0.242,Y -569.130,Z 936.733,A 0.000,B 0.000,C 90.000,E1 347.881} C_DIS
LIN {X 0.123,Y -573.166,Z 936.730,A 0.000,B 0.000,C 90.000,E1 347.297} C_DIS
LIN {X 0.299,Y -578.909,Z 936.725,A 0.000,B 0.000,C 90.000,E1 346.464} C_DIS
LIN {X 0.176,Y -582.424,Z 936.722,A 0.000,B 0.000,C 90.000,E1 345.936} C_DIS
LIN {X 0.226,Y -588.229,Z 936.717,A 0.000,B 0.000,C 90.000,E1 344.991} C_DIS
LIN {X -0.229,Y -593.502,Z 936.712,A 0.000,B 0.000,C 90.000,E1 344.102} C_DIS
LIN {X 0.112,Y -598.421,Z 936.706,A 0.000,B 0.000,C 90.000,E1 343.142} C_DIS
LIN {X 0.238,Y -604.169,Z 936.700,A 0.000,B 0.000,C 90.000,E1 341.945} C_DIS
LIN {X 0.176,Y -607.985,Z 936.695,A 0.000,B 0.000,C 90.000,E1 341.167} C_DIS
LIN {X 0.086,Y -612.772,Z 936.690,A 0.000,B 0.000,C 90.000,E1 340.134} C_DIS
LIN {X 0.269,Y -617.213,Z 936.684,A 0.000,B 0.000,C 90.000,E1 339.082} C_DIS
LIN {X -0.281,Y -621.338,Z 936.678,A 0.000,B 0.000,C 90.000,E1 338.103} C_DIS
LIN {X 0.028,Y -624.332,Z 936.674,A 0.000,B 0.000,C 90.000,E1 337.305} C_DIS
LIN {X -0.200,Y -627.999,Z 936.668,A 0.000,B 0.000,C 90.000,E1 336.305} C_DIS
LIN {X -0.120,Y -631.500,Z 936.663,A 0.000,B 0.000,C 90.000,E1 335.281} C_DIS
LIN {X -0.213,Y -635.559,Z 936.656,A 0.000,B 0.000,C 90.000,E1 334.024} C_DIS
LIN {X 0.034,Y -639.272,Z 936.649,A 0.000,B 0.000,C 90.000,E1 332.743} C_DIS
LIN {X -0.293,Y -641.997,Z 936.643,A 0.000,B 0.000,C 90.000,E1 331.769} C_DIS
LIN {X -0.093,Y -643.916,Z 936.639,A 0.000,B 0.000,C 90.000,E1 331.001} C_DIS
LIN {X 0.103,Y -647.437,Z 936.631,A 0.000,B 0.000,C 90.000,E1 329.488} C_DIS
LIN {X -0.358,Y -649.531,Z 936.625,A 0.000,B 0.000,C 90.000,E1 328.535} C_DIS
LIN {X -0.238,Y -651.355,Z 936.620,A 0.000,B 0.000,C 90.000,E1 327.533} C_DIS
LIN {X 0.172,Y -652.633,Z 936.615,A 0.000,B 0.000,C 90.000,E1 326.755} C_DIS
LIN {X 0.237,Y -654.423,Z 936.609,A 0.000,B 0.000,C 90.000,E1 325.515} C_DIS
LIN {X -0.134,Y -656.183,Z 936.600,A 0.000,B 0.000,C 90.000,E1 324.069} C_DIS
LIN {X 0.278,Y -657.237,Z 936.595,A 0.000,B 0.000,C 90.000,E1 323.050} C_DIS
LIN {X 0.260,Y -658.261,Z 936.588,A 0.000,B 0.000,C 90.000,E1 321.823} C_DIS
LIN {X -0.278,Y -659.832,Z 936.577,A 0.000,B 0.000,C 90.000,E1 319.908} C_DIS
LIN {X 0.121,Y -660.951,Z 936.569,A 0.000,B 0.000,C 90.000,E1 318.405} C_DIS
LIN {X 0.061,Y -662.006,Z 936.562,A 0.000,B 0.000,C 90.000,E1 317.187} C_DIS
LIN {X -0.028,Y -663.184,Z 936.554,A 0.000,B 0.000,C 90.000,E1 315.729} C_DIS
LIN {X -0.119,Y -665.485,Z 936.539,A 0.000,B 0.000,C 90.000,E1 313.056} C_DIS
LIN {X -0.109,Y -666.857,Z 936.531,A 0.000,B 0.000,C 90.000,E1 311.595} C_DIS
LIN {X 0.001,Y -668.405,Z 936.522,A 0.000,B 0.000,C 90.000,E1 309.886} C_DIS
LIN {X 0.071,Y -669.274,Z 936.516,A 0.000,B 0.000,C 90.000,E1 308.910} C_DIS
LIN {X -0.279,Y -670.245,Z 936.510,A 0.000,B 0.000,C 90.000,E1 307.729} C_DIS
LIN {X -0.074,Y -670.835,Z 936.504,A 0.000,B 0.000,C 90.000,E1 306.744} C_DIS
LIN {X 0.017,Y -671.140,Z 936.500,A 0.000,B 0.000,C 90.000,E1 306.011} C_DIS
LIN {X 0.079,Y -671.749,Z 936.489,A 0.000,B 0.000,C 90.000,E1 304.072} C_DIS
LIN {X -0.253,Y -672.835,Z 936.477,A 0.000,B 0.000,C 90.000,E1 301.926} C_DIS
LIN {X -0.295,Y -677.751,Z 936.449,A 0.000,B 0.000,C 90.000,E1 296.873} C_DIS
LIN {X -0.032,Y -680.144,Z 936.441,A 0.000,B 0.000,C 90.000,E1 295.412} C_DIS
LIN {X 0.073,Y -681.996,Z 936.435,A 0.000,B 0.000,C 90.000,E1 294.207} C_DIS
LIN {X -0.213,Y -682.942,Z 936.431,A 0.000,B 0.000,C 90.000,E1 293.515} C_DIS
LIN {X -0.072,Y -683.435,Z 936.428,A 0.000,B 0.000,C 90.000,E1 293.025} C_DIS
LIN {X 0.340,Y -683.665,Z 936.425,A 0.000,B 0.000,C 90.000,E1 292.514} C_DIS
LIN {X -0.143,Y -683.144,Z 936.423,A 0.000,B 0.000,C 90.000,E1 292.078} C_DIS
LIN {X -0.196,Y -682.790,Z 936.421,A 0.000,B 0.000,C 90.000,E1 291.844} C_DIS
LIN {X 0.005,Y -681.681,Z 936.420,A 0.000,B 0.000,C 90.000,E1 291.589} C_DIS
LIN {X 0.104,Y -680.941,Z 936.419,A 0.000,B 0.000,C 90.000,E1 291.461} C_DIS
LIN {X 0.144,Y -678.073,Z 936.417,A 0.000,B 0.000,C 90.000,E1 291.099} C_DIS
LIN {X 0.236,Y -676.877,Z 936.417,A 0.000,B 0.000,C 90.000,E1 290.972} C_DIS
LIN {X 0.133,Y -672.035,Z 936.415,A 0.000,B 0.000,C 90.000,E1 290.663} C_DIS
LIN {X -0.273,Y -664.466,Z 936.412,A 0.000,B 0.000,C 90.000,E1 290.248} C_DIS
LIN {X -0.317,Y -662.191,Z 936.411,A 0.000,B 0.000,C 90.000,E1 290.066} C_DIS
LIN {X -0.356,Y -662.168,Z 936.411,A 0.000,B 0.000,C 90.000,E1 290.066} C_DIS
LIN {X -0.069,Y -661.646,Z 936.410,A 0.000,B 0.000,C 90.000,E1 289.885} C_DIS
LIN {X -0.252,Y -662.383,Z 936.408,A 0.000,B 0.000,C 90.000,E1 289.504} C_DIS
LIN {X 0.011,Y -663.866,Z 936.406,A 0.000,B 0.000,C 90.000,E1 289.087} C_DIS
LIN {X -0.001,Y -666.802,Z 936.403,A 0.000,B 0.000,C 90.000,E1 288.489} C_DIS
LIN {X 0.024,Y -671.290,Z 936.398,A 0.000,B 0.000,C 90.000,E1 287.638} C_DIS
LIN {X 0.018,Y -674.738,Z 936.394,A 0.000,B 0.000,C 90.000,E1 286.913} C_DIS
LIN {X -0.098,Y -676.728,Z 936.391,A 0.000,B 0.000,C 90.000,E1 286.441} C_DIS
LIN {X -0.059,Y -679.160,Z 936.387,A 0.000,B 0.000,C 90.000,E1 285.717} C_DIS
LIN {X -0.144,Y -680.525,Z 936.385,A 0.000,B 0.000,C 90.000,E1 285.245} C_DIS
LIN {X -0.252,Y -682.189,Z 936.381,A 0.000,B 0.000,C 90.000,E1 284.537} C_DIS
LIN {X -0.342,Y -683.637,Z 936.377,A 0.000,B 0.000,C 90.000,E1 283.828} C_DIS
LIN {X 0.248,Y -684.838,Z 936.373,A 0.000,B 0.000,C 90.000,E1 283.063} C_DIS
LIN {X 0.160,Y -686.082,Z 936.367,A 0.000,B 0.000,C 90.000,E1 282.119} C_DIS
LIN {X -0.020,Y -686.511,Z 936.365,A 0.000,B 0.000,C 90.000,E1 281.658} C_DIS
LIN {X -0.057,Y -686.733,Z 936.362,A 0.000,B 0.000,C 90.000,E1 281.186} C_DIS
LIN {X -0.097,Y -686.700,Z 936.360,A 0.000,B 0.000,C 90.000,E1 280.715} C_DIS
LIN {X -0.265,Y -686.303,Z 936.357,A 0.000,B 0.000,C 90.000,E1 280.254} C_DIS
LIN {X -0.288,Y -685.982,Z 936.356,A 0.000,B 0.000,C 90.000,E1 280.018} C_DIS
LIN {X 0.221,Y -685.062,Z 936.353,A 0.000,B 0.000,C 90.000,E1 279.500} C_DIS
LIN {X 0.162,Y -683.675,Z 936.350,A 0.000,B 0.000,C 90.000,E1 279.029} C_DIS
LIN {X -0.016,Y -681.928,Z 936.348,A 0.000,B 0.000,C 90.000,E1 278.568} C_DIS
LIN {X -0.200,Y -679.824,Z 936.345,A 0.000,B 0.000,C 90.000,E1 278.106} C_DIS
LIN {X 0.142,Y -675.668,Z 936.340,A 0.000,B 0.000,C 90.000,E1 277.239} C_DIS
LIN {X -0.238,Y -671.229,Z 936.336,A 0.000,B 0.000,C 90.000,E1 276.429} C_DIS
LIN {X 0.089,Y -667.592,Z 936.332,A 0.000,B 0.000,C 90.000,E1 275.796} C_DIS
LIN {X -0.188,Y -664.296,Z 936.330,A 0.000,B 0.000,C 90.000,E1 275.334} C_DIS
LIN {X 0.080,Y -659.513,Z 936.326,A 0.000,B 0.000,C 90.000,E1 274.702} C_DIS
LIN {X -0.299,Y -655.359,Z 936.323,A 0.000,B 0.000,C 90.000,E1 274.245} C_DIS
LIN {X -0.105,Y -649.598,Z 936.320,A 0.000,B 0.000,C 90.000,E1 273.612} C_DIS
LIN {X 0.233,Y -644.727,Z 936.317,A 0.000,B 0.000,C 90.000,E1 273.094} C_DIS
LIN {X 0.077,Y -638.162,Z 936.314,A 0.000,B 0.000,C 90.000,E1 272.522} C_DIS
LIN {X -0.304,Y -631.306,Z 936.311,A 0.000,B 0.000,C 90.000,E1 272.007} C_DIS
LIN {X -0.263,Y -624.011,Z 936.308,A 0.000,B 0.000,C 90.000,E1 271.489} C_DIS
LIN {X -0.254,Y -617.896,Z 936.306,A 0.000,B 0.000,C 90.000,E1 271.088} C_DIS
LIN {X 0.023,Y -611.668,Z 936.304,A 0.000,B 0.000,C 90.000,E1 270.688} C_DIS
LIN {X 0.173,Y -603.396,Z 936.301,A 0.000,B 0.000,C 90.000,E1 270.229} C_DIS
LIN {X -0.014,Y -598.309,Z 936.300,A 0.000,B 0.000,C 90.000,E1 270.000} C_DIS
LIN {X -0.135,Y -591.406,Z 936.298,A 0.000,B 0.000,C 90.000,E1 269.714} C_DIS
LIN {X 0.008,Y -583.902,Z 936.297,A 0.000,B 0.000,C 90.000,E1 269.427} C_DIS
LIN {X 0.018,Y -578.121,Z 936.296,A 0.000,B 0.000,C 90.000,E1 269.255} C_DIS
LIN {X -0.104,Y -570.282,Z 936.295,A 0.000,B 0.000,C 90.000,E1 269.083} C_DIS
LIN {X -0.022,Y -564.613,Z 936.294,A 0.000,B 0.000,C 90.000,E1 268.969} C_DIS
LIN {X -0.139,Y -558.442,Z 936.294,A 0.000,B 0.000,C 90.000,E1 268.912} C_DIS
LIN {X 0.012,Y -551.959,Z 936.294,A 0.000,B 0.000,C 90.000,E1 268.854} C_DIS
LIN {X -0.256,Y -550.472,Z 936.294,A 0.000,B 0.000,C 90.000,E1 268.854} C_DIS
LIN {X 0.261,Y -550.419,Z 936.294,A 0.000,B 0.000,C 90.000,E1 268.797} C_DIS
LIN {X 0.103,Y -549.082,Z 936.292,A 0.000,B 0.000,C 90.000,E1 268.625} C_DIS
LIN {X -0.092,Y -545.412,Z 936.290,A 0.000,B 0.000,C 90.000,E1 268.224} C_DIS
LIN {X -0.117,Y -544.058,Z 936.289,A 0.000,B 0.000,C 90.000,E1 268.108} C_DIS
LIN {X -0.159,Y -544.003,Z 936.289,A 0.000,B 0.000,C 90.000,E1 268.108} C_DIS
LIN {X 0.001,Y -543.157,Z 936.287,A 0.000,B 0.000,C 90.000,E1 267.650} C_DIS
LIN {X -0.040,Y -540.434,Z 936.270,A 0.000,B 0.000,C 90.000,E1 264.546} C_DIS
LIN {X 0.162,Y -539.100,Z 936.259,A 0.000,B 0.000,C 90.000,E1 262.534} C_DIS
LIN {X -0.192,Y -538.331,Z 936.252,A 0.000,B 0.000,C 90.000,E1 261.432} C_DIS
LIN {X 0.003,Y -537.633,Z 936.248,A 0.000,B 0.000,C 90.000,E1 260.557} C_DIS
LIN {X 0.040,Y -537.016,Z 936.244,A 0.000,B 0.000,C 90.000,E1 259.982} C_DIS
LIN {X -0.244,Y -535.412,Z 936.238,A 0.000,B 0.000,C 90.000,E1 258.870} C_DIS
LIN {X -0.099,Y -531.295,Z 936.221,A 0.000,B 0.000,C 90.000,E1 255.700} C_DIS
LIN {X -0.164,Y -529.590,Z 936.213,A 0.000,B 0.000,C 90.000,E1 254.267} C_DIS
LIN {X 0.060,Y -528.580,Z 936.208,A 0.000,B 0.000,C 90.000,E1 253.378} C_DIS
LIN {X -0.058,Y -526.829,Z 936.200,A 0.000,B 0.000,C 90.000,E1 251.945} C_DIS
LIN {X 0.114,Y -524.607,Z 936.190,A 0.000,B 0.000,C 90.000,E1 250.188} C_DIS
LIN {X -0.072,Y -522.361,Z 936.180,A 0.000,B 0.000,C 90.000,E1 248.465} C_DIS
LIN {X 0.073,Y -520.837,Z 936.174,A 0.000,B 0.000,C 90.000,E1 247.283} C_DIS
LIN {X -0.134,Y -518.655,Z 936.166,A 0.000,B 0.000,C 90.000,E1 245.845} C_DIS
LIN {X -0.052,Y -516.795,Z 936.159,A 0.000,B 0.000,C 90.000,E1 244.665} C_DIS
LIN {X -0.248,Y -514.989,Z 936.153,A 0.000,B 0.000,C 90.000,E1 243.512} C_DIS
LIN {X -0.121,Y -512.586,Z 936.145,A 0.000,B 0.000,C 90.000,E1 242.025} C_DIS
LIN {X -0.046,Y -510.131,Z 936.136,A 0.000,B 0.000,C 90.000,E1 240.539} C_DIS
LIN {X 0.154,Y -508.049,Z 936.130,A 0.000,B 0.000,C 90.000,E1 239.331} C_DIS
LIN {X 0.060,Y -505.771,Z 936.123,A 0.000,B 0.000,C 90.000,E1 238.152} C_DIS
LIN {X 0.152,Y -503.907,Z 936.118,A 0.000,B 0.000,C 90.000,E1 237.248} C_DIS
LIN {X 0.006,Y -499.802,Z 936.108,A 0.000,B 0.000,C 90.000,E1 235.468} C_DIS
LIN {X 0.201,Y -494.999,Z 936.096,A 0.000,B 0.000,C 90.000,E1 233.336} C_DIS
LIN {X 0.031,Y -491.087,Z 936.086,A 0.000,B 0.000,C 90.000,E1 231.537} C_DIS
LIN {X 0.238,Y -487.695,Z 936.078,A 0.000,B 0.000,C 90.000,E1 229.989} C_DIS
LIN {X 0.141,Y -483.491,Z 936.068,A 0.000,B 0.000,C 90.000,E1 228.162} C_DIS
LIN {X -0.284,Y -478.634,Z 936.056,A 0.000,B 0.000,C 90.000,E1 226.053} C_DIS
LIN {X -0.274,Y -474.555,Z 936.045,A 0.000,B 0.000,C 90.000,E1 224.190} C_DIS
LIN {X -0.111,Y -471.098,Z 936.037,A 0.000,B 0.000,C 90.000,E1 222.609} C_DIS
LIN {X 0.020,Y -467.605,Z 936.028,A 0.000,B 0.000,C 90.000,E1 221.024} C_DIS
LIN {X -0.070,Y -462.148,Z 936.014,A 0.000,B 0.000,C 90.000,E1 218.508} C_DIS
LIN {X -0.072,Y -459.381,Z 936.007,A 0.000,B 0.000,C 90.000,E1 217.237} C_DIS
LIN {X -0.105,Y -455.951,Z 935.998,A 0.000,B 0.000,C 90.000,E1 215.644} C_DIS
LIN {X -0.108,Y -452.460,Z 935.989,A 0.000,B 0.000,C 90.000,E1 214.040} C_DIS
LIN {X 0.108,Y -447.367,Z 935.977,A 0.000,B 0.000,C 90.000,E1 211.750} C_DIS
LIN {X 0.009,Y -444.547,Z 935.969,A 0.000,B 0.000,C 90.000,E1 210.463} C_DIS
LIN {X 0.161,Y -439.590,Z 935.957,A 0.000,B 0.000,C 90.000,E1 208.153} C_DIS
LIN {X -0.108,Y -436.801,Z 935.949,A 0.000,B 0.000,C 90.000,E1 206.873} C_DIS
LIN {X -0.196,Y -432.373,Z 935.938,A 0.000,B 0.000,C 90.000,E1 204.899} C_DIS
LIN {X -0.174,Y -428.012,Z 935.927,A 0.000,B 0.000,C 90.000,E1 202.898} C_DIS
LIN {X -0.024,Y -423.531,Z 935.916,A 0.000,B 0.000,C 90.000,E1 200.865} C_DIS
LIN {X -0.025,Y -417.152,Z 935.899,A 0.000,B 0.000,C 90.000,E1 197.819} C_DIS
LIN {X 0.222,Y -413.801,Z 935.890,A 0.000,B 0.000,C 90.000,E1 196.079} C_DIS
LIN {X 0.155,Y -411.027,Z 935.882,A 0.000,B 0.000,C 90.000,E1 194.717} C_DIS
LIN {X -0.205,Y -405.396,Z 935.867,A 0.000,B 0.000,C 90.000,E1 192.007} C_DIS
LIN {X -0.100,Y -402.053,Z 935.857,A 0.000,B 0.000,C 90.000,E1 190.254} C_DIS
LIN {X -0.137,Y -398.692,Z 935.847,A 0.000,B 0.000,C 90.000,E1 188.511} C_DIS
LIN {X 0.060,Y -394.635,Z 935.836,A 0.000,B 0.000,C 90.000,E1 186.372} C_DIS
LIN {X -0.075,Y -389.296,Z 935.820,A 0.000,B 0.000,C 90.000,E1 183.555} C_DIS
LIN {X 0.139,Y -383.560,Z 935.800,A 0.000,B 0.000,C 90.000,E1 179.943} C_DIS
LIN {X 0.189,Y -382.386,Z 935.794,A 0.000,B 0.000,C 90.000,E1 178.854} C_DIS
LIN {X -0.145,Y -381.794,Z 935.788,A 0.000,B 0.000,C 90.000,E1 177.822} C_DIS
LIN {X -0.037,Y -382.010,Z 935.783,A 0.000,B 0.000,C 90.000,E1 177.020} C_DIS
LIN {X 0.126,Y -382.778,Z 935.779,A 0.000,B 0.000,C 90.000,E1 176.274} C_DIS
LIN {X -0.085,Y -384.611,Z 935.775,A 0.000,B 0.000,C 90.000,E1 175.584} C_DIS
LIN {X -0.203,Y -386.190,Z 935.773,A 0.000,B 0.000,C 90.000,E1 175.241} C_DIS
LIN {X 0.099,Y -389.385,Z 935.771,A 0.000,B 0.000,C 90.000,E1 174.666} C_DIS
LIN {X 0.040,Y -393.806,Z 935.768,A 0.000,B 0.000,C 90.000,E1 174.147} C_DIS
LIN {X 0.087,Y -395.378,Z 935.767,A 0.000,B 0.000,C 90.000,E1 173.970} C_DIS
LIN {X -0.086,Y -402.864,Z 935.763,A 0.000,B 0.000,C 90.000,E1 173.337} C_DIS
LIN {X 0.002,Y -417.502,Z 935.757,A 0.000,B 0.000,C 90.000,E1 172.186} C_DIS
LIN {X -0.061,Y -431.426,Z 935.750,A 0.000,B 0.000,C 90.000,E1 171.084} C_DIS
LIN {X -0.190,Y -440.676,Z 935.746,A 0.000,B 0.000,C 90.000,E1 170.330} C_DIS
LIN {X 0.187,Y -450.475,Z 935.741,A 0.000,B 0.000,C 90.000,E1 169.398} C_DIS
LIN {X -0.057,Y -460.593,Z 935.736,A 0.000,B 0.000,C 90.000,E1 168.465} C_DIS
LIN {X 0.164,Y -466.116,Z 935.733,A 0.000,B 0.000,C 90.000,E1 167.881} C_DIS
LIN {X 0.163,Y -474.183,Z 935.728,A 0.000,B 0.000,C 90.000,E1 166.992} C_DIS
LIN {X -0.028,Y -479.489,Z 935.725,A 0.000,B 0.000,C 90.000,E1 166.408} C_DIS
LIN {X 0.215,Y -487.046,Z 935.719,A 0.000,B 0.000,C 90.000,E1 165.463} C_DIS
LIN {X -0.268,Y -493.247,Z 935.715,A 0.000,B 0.000,C 90.000,E1 164.755} C_DIS
LIN {X 0.129,Y -497.737,Z 935.712,A 0.000,B 0.000,C 90.000,E1 164.102} C_DIS
LIN {X -0.203,Y -505.272,Z 935.706,A 0.000,B 0.000,C 90.000,E1 163.087} C_DIS
LIN {X 0.006,Y -513.325,Z 935.699,A 0.000,B 0.000,C 90.000,E1 161.873} C_DIS
LIN {X 0.209,Y -519.265,Z 935.694,A 0.000,B 0.000,C 90.000,E1 160.967} C_DIS
LIN {X 0.134,Y -525.829,Z 935.689,A 0.000,B 0.000,C 90.000,E1 159.953} C_DIS
LIN {X 0.203,Y -534.134,Z 935.682,A 0.000,B 0.000,C 90.000,E1 158.646} C_DIS
LIN {X -0.008,Y -540.258,Z 935.676,A 0.000,B 0.000,C 90.000,E1 157.667} C_DIS
LIN {X 0.065,Y -549.619,Z 935.667,A 0.000,B 0.000,C 90.000,E1 156.102} C_DIS
LIN {X -0.136,Y -554.433,Z 935.663,A 0.000,B 0.000,C 90.000,E1 155.281} C_DIS
LIN {X 0.007,Y -560.544,Z 935.656,A 0.000,B 0.000,C 90.000,E1 154.152} C_DIS
LIN {X 0.071,Y -565.592,Z 935.651,A 0.000,B 0.000,C 90.000,E1 153.179} C_DIS
LIN {X -0.148,Y -570.888,Z 935.645,A 0.000,B 0.000,C 90.000,E1 152.103} C_DIS
LIN {X -0.035,Y -576.043,Z 935.639,A 0.000,B 0.000,C 90.000,E1 151.001} C_DIS
LIN {X -0.215,Y -579.529,Z 935.634,A 0.000,B 0.000,C 90.000,E1 150.205} C_DIS
